DATA_BLOCK "LT"   // DB201
{ S7_Optimized_Access := 'FALSE' }
VERSION : 0.0
// --------------------------------------------------------------------------------
//     program     :    LT
//     description :    define all LT values       
//     name        :    G. Eibelsh鋟ser
//     date        :    26.10.2007
// 
//     revision    :   
//     name        :   
//     date        :    
// 
//                     (c)PVA TePla AG       
//     --------------------------------------------------------------------------------
   VAR
      MOD_AUTO : Bool;   // word 0
      MOD_MANUAL : Bool;
      MOD_SERVICE : Bool;
      MOD_SEMI_AUTO : Bool;
      MOD_START : Bool;
      MOD_CONTINUE : Bool;
      MOD_STOP : Bool;
      SPARE_0_7 : Bool;
      MOD_PUMP_DOWN : Bool;
      MOD_MELTING : Bool;
      MOD_DIP : Bool;
      MOD_NECK : Bool;
      MOD_SHOULDER : Bool;
      MOD_BODY : Bool;
      MOD_ENDCONE : Bool;
      MOD_REMOVAL : Bool;
      MOD_SHUT_DOWN : Bool;   // word 1
      MOD_EMG : Bool;
      SPARE_2_2 : Bool;
      SPARE_2_3 : Bool;
      SPARE_2_4 : Bool;
      SPARE_2_5 : Bool;
      SPARE_2_6 : Bool;
      SPARE_2_7 : Bool;
      SMI_XT_SPD_ON : Bool;
      SMI_XT_ROT_ON : Bool;
      SMI_CR_SPD_ON : Bool;
      SMI_CR_ROT_ON : Bool;
      SMI_HTR_1_ON : Bool;
      SMI_HTR_2_ON : Bool;
      SMI_GAS_FLW_ON : Bool;
      SMI_GAS_PRS_ON : Bool;
      SMI_SI_FDR_ON : Bool;   // word 2
      SMI_DOP_FDR_ON : Bool;
      SMI_MAG_ON : Bool;
      SMI_CR_SPD_COF_ON : Bool;
      SMI_MOB_FDR_ON : Bool;
      SPARE_4_5 : Bool;
      SPARE_4_6 : Bool;
      SPARE_4_7 : Bool;
      XT_LFT_UP : Bool;
      XT_LFT_DN : Bool;
      XT_LFT_FST : Bool;
      XT_ROT_CW : Bool;
      XT_ROT_CCW : Bool;
      XT_ROT_OFF : Bool;
      XT_LFT_OFF : Bool;
      CCZ_OP_ON : Bool;
      CR_LFT_UP : Bool;   // word 3
      CR_LFT_DN : Bool;
      CR_LFT_FST : Bool;
      CR_ROT_CW : Bool;
      CR_ROT_CCW : Bool;
      CR_ROT_OFF : Bool;
      CR_LFT_OFF : Bool;
      SPARE_6_7 : Bool;
      HTR_1_ON : Bool;
      HTR_2_ON : Bool;
      MAG_ON : Bool;
      P2_ON : Bool;
      SI_CRG_WGT_VALID : Bool;
      MAG_STBY_ON : Bool;
      DBL_ALM_SND : Bool;
      CTL_AV_CRUC_ROT_ON : Bool;
      CTL_DIA_ON : Bool;   // word 4
      CTL_GRO_ON : Bool;
      CTL_LVL_ON : Bool;
      CTL_AV_SPD_ON : Bool;
      CTL_HTR_1_TMP_ON : Bool;
      CTL_MELT_TMP_1_ON : Bool;
      CTL_HTR_2_TMP_ON : Bool;
      CTL_MELT_TMP_2_ON : Bool;
      CTL_PRS_ON : Bool;
      V1_OPEN_REQ : Bool;
      V1_CLOSE_REQ : Bool;
      V7_OPEN : Bool;
      V7_CLOSE : Bool;
      V2_1_SEL : Bool;
      V2_2_SEL : Bool;
      V2_X_SEL : Bool;
      V1_OPEN : Bool;   // word 5
      V2_1_OPEN : Bool;
      V3_OPEN : Bool;
      V4_OPEN : Bool;
      V5_OPEN : Bool;
      V6_OPEN : Bool;
      V8_OPEN : Bool;
      V11_OP : Bool;
      V12_OPEN : Bool;
      V2_2_OPEN : Bool;
      V9_1_OPEN : Bool;
      V9_2_OPEN : Bool;
      V1_LS_OPEN : Bool;
      V1_LS_CLOSE : Bool;
      P1_ON : Bool;
      P3_ON : Bool;
      MCC_ON : Bool;   // word 6
      MCC_TST_ON : Bool;
      LSR_ON : Bool;
      LSR_OFF : Bool;
      V16_1_OPEN : Bool;
      V16_2_OPEN : Bool;
      V21_OPEN : Bool;
      CAM_RST_THR_ADJ_ENB : Bool;
      CAM_OFF : Bool;
      CAM_MLT : Bool;
      CAM_DIP : Bool;
      CAM_DIA : Bool;
      CAM_INIT : Bool;
      CAM_SEL_1 : Bool;
      CAM_SEL_2 : Bool;
      CAM_RST_THR_ADJ_DIS : Bool;
      PNBDY : Bool;   // word 7
      BYRST : Bool;
      SUTDN : Bool;
      LEN2_CALC : Bool;
      PMELT : Bool;
      XT_MELT_CONTACT : Bool;
      ALARM : Bool;
      VAC_FNC : Bool;
      VAC_GAT : Bool;
      CLF_APS : Bool;
      CGT_APS : Bool;
      OP_CALL_ON : Bool;
      OP_CALL_ALM : Bool;
      LSR_FIL_LOW : Bool;
      LSR_FIL_HI : Bool;
      LSR_LVL_ABV_REF : Bool;
      FDR_HOP_CON : Bool;   // word 8
      FDR_APS : Bool;
      FDR_LS_TUBE_IN : Bool;
      FDR_LS_TUBE_OUT : Bool;
      FDR_TUBE_DRV_IN : Bool;
      FDR_TUBE_DRV_OUT : Bool;
      FDR_TUBE_DRV_OFF : Bool;
      FDR_FLP_CTL_ON : Bool;
      FDR_FLP_CTL_OFF : Bool;
      XT_DRP_OUT_PRT_OP : Bool;
      XT_DRP_OUT_PRT_CL : Bool;
      XT_DRP_OUT_PRT_ENB : Bool;
      V11_CL : Bool;
      V3_2_OP : Bool;
      V24_OP : Bool;
      PRC_RUN_DONE : Bool;
      CAM_ISP_ON : Bool;   // word 9
      EMG_MOD_REQ : Bool;
      MA_NOT_AVL : Bool;
      NOT_ACKN_ALM : Bool;
      V13_OPEN : Bool;
      V14_OPEN : Bool;
      V15_OPEN : Bool;
      V17_OPEN : Bool;
      V18_OPEN : Bool;
      V19_OPEN : Bool;
      V20_OPEN : Bool;
      V22_OPEN : Bool;
      V23_OPEN : Bool;
      VAC_LINE_IS_OPEN : Bool;
      AUX_FIL_ENB : Bool;
      CAM_PRD_1_SEL : Bool;
      CAM_PRD_2_SEL : Bool;   // word 10
      V25_OPEN : Bool;
      SI_FIL_FSH_SEQ_ON : Bool;
      EDIT_INGOT_ID : Bool;
      EDIT_CARRIER_ID : Bool;
      ENB_LOADING : Bool;
      SMI_GAP_ON : Bool;
      LSR_SEN_PWR_ON : Bool;
      RST_SIHI_PU : Bool;
      RST_HTR_1_PWR_SPL : Bool;
      RST_HTR_2_PWR_SPL : Bool;
      AUTO_OP_CALL : Bool;
      EXT_ACQ_TRG_ON : Bool;
      CAM_CAL : Bool;
      SPARE_21_6 : Bool;
      SPARE_21_7 : Bool;
      CTL_MLT_DRIFT_ON : Bool;   // word 11
      RST_MLT_LVL : Bool;
      MSR_MLT_VIB_ON : Bool;
      SPARE_22_3 : Bool;
      SPARE_22_4 : Bool;
      SPARE_22_5 : Bool;
      SPARE_22_6 : Bool;
      SPARE_22_7 : Bool;
      TEST_CTRL_ON : Bool;
      TEST_CTRL_RST : Bool;
      EMG_ON : Bool;
      SPARE_23_3 : Bool;
      SPARE_23_4 : Bool;
      SPARE_23_5 : Bool;
      BY_FIL_APS : Bool;
      FIL_APS : Bool;
      V3_0_OPEN : Bool;   // word 12
      V3_1_OPEN : Bool;
      XT_LFT_REF_RUN : Bool;
      CR_LFT_REF_RUN : Bool;
      XT_LFT_REF_DONE : Bool;
      CR_LFT_REF_DONE : Bool;
      XT_LFT_REL_LS : Bool;
      CR_LFT_REL_LS : Bool;
      MOB_FDR_IN_POS : Bool;
      MOB_FDR_DCK_ATV : Bool;
      MOB_FDR_UDCK_ATV : Bool;
      MOB_FDR_DCK_DONE : Bool;
      MOB_FDR_UDCK_DONE : Bool;
      MOB_FDR_CH_FDG_POS : Bool;
      ACC_OVP_TEST_ENB : Bool;
      ACC_OVP_OK : Bool;
      MOB_FDR_MVE_IN_SEQ_ON : Bool;   // word 13
      MOB_FDR_MVE_OUT_SEQ_ON : Bool;
      MOB_FDR_MVE_SEQ_ARB : Bool;
      MOB_FDR_VIB_ON : Bool;
      MOB_FDR_CH_HOME_POS : Bool;
      MOB_FDR_TUBE_HOME_POS : Bool;
      MOB_FDR_TUBE_FCH_POS : Bool;
      MOB_FDR_TUBE_FDG_POS : Bool;
      MOB_FDR_EL_CON_DONE : Bool;
      ACC_OVP_TEST_ON : Bool;
      ACC_SC_WTR_STR_ON : Bool;
      ACC_SC_WTR_STR_ENB : Bool;
      SHOW_HTR_1_TRG_TMP : Bool;
      SHOW_XT_RMV_BTN : Bool;
      ENB_KEY_NEXT_MLT_STEP : Bool;
      CTL_FDG_RTE_ON : Bool;
      MOB_FDR_SRV_ON : Bool;
      MOB_FDR_TUBE_UP : Bool;
      MOB_FDR_TUBE_DN : Bool;
      MOB_FDR_TUBE_STOP : Bool;
      MOB_FDR_CH_SW_R : Bool;
      MOB_FDR_CH_SW_L : Bool;
      MOB_FDR_CH_SW_STOP : Bool;
      SH_MLT_LVL_SFT_RUN : Bool;
      ARR_ID_PD : Bool;
      ARR_PD_ID : Bool;
      ARR_PD_ME : Bool;
      ARR_EC_SD : Bool;
      ARR_BY_RE : Bool;
      ARR_EC_RE : Bool;
      ARR_RE_DI : Bool;
      TCH_HOOK_1_ABV : Bool;
      TCH_HOOK_2_ABV : Bool;   // word 15
      TCH_HOOK_3_ABV : Bool;
      TCH_HOOK_4_ABV : Bool;
      TCH_HOOK_1_BLW : Bool;
      TCH_HOOK_2_BLW : Bool;
      TCH_HOOK_3_BLW : Bool;
      TCH_HOOK_4_BLW : Bool;
      GCH_SWD_IN : Bool;
      GCH_SWD_OUT : Bool;
      TCH_CON_GCH : Bool;
      CUF_CLP_LS_SWV_IN_1 : Bool;
      CUF_CLP_LS_SWV_OUT_1 : Bool;
      CUF_CLP_LS_SWV_IN_2 : Bool;
      CUF_CLP_LS_SWV_OUT_2 : Bool;
      HND_LFT_UP : Bool;
      HND_LFT_DN : Bool;
      GCH_SWV_IN : Bool;   // word 16
      GCH_SWV_OUT : Bool;
      MAG_RAI_ON : Bool;
      MAG_LOW_ON : Bool;
      CTL_GAP_ON : Bool;
      SPARE_32_5 : Bool;
      SPARE_32_6 : Bool;
      SPARE_32_7 : Bool;
      SPARE_33_0 : Bool;
      SPARE_33_1 : Bool;
      SPARE_33_2 : Bool;
      SPARE_33_3 : Bool;
      SPARE_33_4 : Bool;
      SPARE_33_5 : Bool;
      SPARE_33_6 : Bool;
      SPARE_33_7 : Bool;
      SPARE : Array[34..63] of Byte;
      XT_HDL_SEQ_MOD : Bool;
      XT_HDL_SEQ_XT_OUT : Bool;
      XT_HDL_SEQ_LD_CRU : Bool;
      XT_HDL_SEQ_HDL_HZ : Bool;
      XT_HDL_OP_CONT : Bool;
      ABORT_FIL_CLN : Bool;
      MLT_GAP_SEARCH : Bool;
      V7_CLN : Bool;
      V7_SW_OUT : Bool;
      V7_SW_IN : Bool;
      V7_LFT_UP : Bool;
      V7_LFT_DN : Bool;
      V7_LFT_UP_REL : Bool;
      V7_LFT_DN_REL : Bool;
      V7_SW_OUT_REL : Bool;
      V7_SW_IN_REL : Bool;
      BEL_LFT_UP_REL : Bool;   // Freigabe
      BEL_LFT_DN_REL : Bool;
      GCH_LFT_UP_REL : Bool;
      GCH_LFT_DN_REL : Bool;
      GCH_SW_OUT_REL : Bool;
      GCH_SW_IN_REL : Bool;
      GCH_SW_LOCKED : Bool;
      TCH_LFT_UP_REL : Bool;
      TCH_LFT_DN_REL : Bool;
      TCH_SW_OUT_REL : Bool;
      TCH_SW_IN_REL : Bool;
      TCH_SW_LOCKED : Bool;
      TCH_TILT_0_REL : Bool;
      TCH_TILT_30_REL : Bool;
      TEC_FLG_LFT_UP_REL : Bool;
      TEC_FLG_LFT_DN_REL : Bool;
      TEC_FLG_SW_OUT_REL : Bool;
      TEC_FLG_SW_IN_REL : Bool;
      TEC_FLG_SW_UNLOCK : Bool;
      UP_FCH_SW_OUT_REL : Bool;
      UP_FCH_SW_IN_REL : Bool;
      UP_FCH_SW_UNLOCK : Bool;
      LO_FCH_SW_OUT_REL : Bool;
      LO_FCH_SW_IN_REL : Bool;
      LO_FCH_SW_UNLOCK : Bool;
      FCH_LFT_UP_REL : Bool;
      FCH_LFT_DN_REL : Bool;
      FCH_HOOK_WORK_REL : Bool;
      FCH_HOOK_HOME_REL : Bool;
      MAG_LFT_UP_REL : Bool;
      MAG_LFT_DN_REL : Bool;
      RESET_ERR_HTR_ETH : Bool;
      SPARE_70_0 : Bool;
      SPARE_70_1 : Bool;
      SPARE_70_2 : Bool;
      SPARE_70_3 : Bool;
      SPARE_70_4 : Bool;
      SPARE_70_5 : Bool;
      SPARE_70_6 : Bool;
      SPARE_70_7 : Bool;
      BEL_LFT_UP : Bool;   // light signals for drives
      BEL_LFT_DN : Bool;
      GCH_LFT_UP : Bool;
      GCH_LFT_DN : Bool;
      TCH_LFT_UP : Bool;
      TCH_LFT_DN : Bool;
      TCH_TILT_0 : Bool;
      TCH_TILT_30 : Bool;
      TEC_FLG_LFT_UP : Bool;
      TEC_FLG_LFT_DN : Bool;
      FCH_LFT_UP : Bool;
      FCH_LFT_DN : Bool;
      MAG_LFT_UP : Bool;
      MAG_LFT_DN : Bool;
      SPARE_72_6 : Bool;
      SPARE_72_7 : Bool;
      GCH_BEL_UP : Bool;   // signals for position of parts
      GCH_BEL_DN : Bool;
      GCH_UP : Bool;
      GCH_DN : Bool;
      GCH_IN : Bool;
      GCH_CLN : Bool;
      GCH_OUT : Bool;
      TCH_UP : Bool;
      TCH_DN : Bool;
      TCH_IN : Bool;
      TCH_CLN : Bool;
      TCH_OUT : Bool;
      TCH_TILT_POS_0 : Bool;
      TCH_TILT_POS_30 : Bool;
      TEC_FLG_SW_OUT : Bool;
      TEC_FLG_SW_IN : Bool;
      UP_FCH_SW_OUT : Bool;
      UP_FCH_SW_IN : Bool;
      LO_FCH_SW_OUT : Bool;
      LO_FCH_SW_IN : Bool;
      GCH_SW_UNLOCK : Bool;
      TCH_SW_UNLOCK : Bool;
      FCH_HOOK_WORK : Bool;
      FCH_HOOK_HOME : Bool;
      MAG_UP : Bool;
      MAG_DN : Bool;
      SPARE_76_2 : Bool;
      SPARE_76_3 : Bool;
      XT_HDL_LFT_DN_REL : Bool;
      XT_HDL_LFT_UP_REL : Bool;
      XT_HDL_SW_OUT_REL : Bool;
      XT_HDL_SW_IN_REL : Bool;
      XT_SLID_FW_REL : Bool;
      XT_SLID_BW_REL : Bool;
      XT_TILT_90_REL : Bool;
      XT_TILT_75_REL : Bool;
      SPARE_77_4 : Bool;
      SPARE_77_5 : Bool;
      SPARE_77_6 : Bool;
      SPARE_77_7 : Bool;
      XT_HDL_LFT_DN : Bool;
      XT_HDL_LFT_UP : Bool;
      XT_HDL_SW_OUT : Bool;
      XT_HDL_SW_IN : Bool;
      XT_SLID_BW : Bool;
      XT_SLID_MID : Bool;
      XT_SLID_FW : Bool;
      XT_TILT_90 : Bool;
      XT_TILT_75 : Bool;
      UP_XT_CLP_CL : Bool;
      UP_XT_CLP_OP : Bool;
      LO_XT_CLP_CL : Bool;
      LO_XT_CLP_OP : Bool;
      SPARE_79_5 : Bool;
      LS_XT_HDL_SW_OUT : Bool;
      LS_XT_HDL_SW_IN : Bool;
      LS_XT_SLID_BW : Bool;
      LS_XT_SLID_MID : Bool;
      LS_XT_SLID_FW : Bool;
      LS_XT_TILT_90 : Bool;
      LS_XT_TILT_75 : Bool;
      LS_UP_XT_CLP_CL : Bool;
      LS_UP_XT_CLP_OP : Bool;
      LS_LO_XT_CLP_CL : Bool;
      LS_LO_XT_CLP_OP : Bool;
      LS_XT_DRP_OUT_PRT_CL : Bool;
      LS_XT_DRP_OUT_PRT_OP : Bool;
      XT_DRP_OUT_PRT_REL : Bool;
      UP_XT_CLP_CL_REL : Bool;
      UP_XT_CLP_OP_REL : Bool;
      LO_XT_CLP_CL_REL : Bool;
      LO_XT_CLP_OP_REL : Bool;
      XT_HDL_LFT_REF_RUN : Bool;
      XT_HDL_LFT_REF_DONE : Bool;
      XT_HDL_SW_REF_RUN : Bool;
      XT_HDL_SW_REF_DONE : Bool;
      XT_HDL_SW_LOCKED : Bool;
      XT_HDL_SW_UNLOCKED : Bool;
      LS_UP_XT_CLP_PLATE : Bool;
      XT_HDL_CLP_OP_CONT : Bool;
      XT_HDL_CUT_OP_CONT : Bool;
      HOI_TOOL_INST : Bool;
      HOI_TOOL_CRU_INS : Bool;
      LD_CRU_OP_CONT : Bool;
      LD_CRU_FIN : Bool;
      HOI_TOOL_UNIS : Bool;
      HOI_TOOL_HZ_INS : Bool;
      LD_HZ_OP_CONT : Bool;
      LD_HZ_FIN : Bool;
      SI_FIL_RDY : Bool;
      MP_SERVICE : Bool;
      V2_11_OPEN : Bool;
      V1_1_OPEN : Bool;
      V3_3_OPEN : Bool;
      V3_4_OPEN : Bool;
      V22_1_OPEN : Bool;
      SPARE_OP : Array[82..127] of Byte;
   END_VAR
BEGIN
END_DATA_BLOCK

DATA_BLOCK "DIS"   // DB202
{ S7_Optimized_Access := 'FALSE' }
VERSION : 0.0
// --------------------------------------------------------------------------------
//     program     :    DIS
//     description :    define all DIS values       
//     name        :    G. Eibelsh鋟ser
//     date        :    26.10.2007
// 
//     revision    :
//     name        :
//     date        :    
//                     (c)PVA TePla AG       
//     --------------------------------------------------------------------------------
   VAR
      SET_XT_SPD : Real;   // dword 0
      ACT_XT_SPD : Real;
      SET_XT_ROT : Real;
      ACT_XT_ROT : Real;
      ACT_XT_POS : Real;
      SET_CR_SPD : Real;
      ACT_CR_SPD : Real;
      SET_CR_ROT : Real;
      ACT_CR_ROT : Real;   // dword 32
      ACT_CR_POS : Real;
      SET_HTR_1_PWR : Real;
      ACT_HTR_1_PWR : Real;
      SET_HTR_1_TMP : Real;
      ACT_HTR_1_TMP : Real;
      ACT_HTR_1_AV_TMP : Real;
      ACT_HTR_1_CUR : Real;
      ACT_HTR_1_VLT : Real;   // dword 64
      ACT_HTR_1_RES : Real;
      SET_HTR_1_TMP_INC : Real;
      ACT_HTR_1_TMP_INC : Real;
      SET_HTR_2_PWR : Real;
      ACT_HTR_2_PWR : Real;
      SET_HTR_2_TMP : Real;
      ACT_HTR_2_TMP : Real;
      ACT_HTR_2_AV_TMP : Real;   // dword 96
      ACT_HTR_2_CUR : Real;
      ACT_HTR_2_VLT : Real;
      ACT_HTR_2_RES : Real;
      SET_HTR_2_PWR_INC : Real;
      ACT_HTR_2_PWR_INC : Real;
      SET_MAG_1_CUR : Real;
      ACT_MAG_1_CUR : Real;
      ACT_MAG_1_VLT : Real;   // dword 128
      ACT_MAG_1_RES : Real;
      SET_MAG_2_CUR : Real;
      ACT_MAG_2_CUR : Real;
      ACT_MAG_2_VLT : Real;
      ACT_MAG_2_RES : Real;
      SET_GAS_1_FLW : Real;
      ACT_GAS_1_FLW : Real;
      SET_GAS_2_FLW : Real;   // dword 160
      ACT_GAS_2_FLW : Real;
      SET_PRS_FNC : Real;
      HTR_1_TMP_SET_PHA_STR : Real;   // heater 1 temperature setpoint at phase start
      HTR_2_PWR_SET_PHA_STR : Real;   // heater 2 power setpoint at phase start
      ACT_TOT_XT_LGH : Real;   // actual total crystal lenght (neck, shoulder, body, endcone)
      ACT_PRS_DROP_FDR : Real;
      ACT_PRS_CLF : Real;   // actual pressure furnace
      ACT_PRS_CGT : Real;   // dword 192 // actual pressure gate
      ACT_PRS_FDR : Real;   // actual pressure feeder
      SET_CTL_VALVE_POS : Real;
      ACT_LEAKR_FNC : Real;
      ACT_LEAKR_FDR : Real;
      SET_XT_DIA : Real;
      ACT_XT_DIA : Real;
      SET_XT_AV_SPD : Real;
      ACT_XT_AV_SPD : Real;   // dword 224
      SET_LSR_MLT_LVL : Real;
      ACT_LSR_MLT_LVL : Real;
      SET_XTAL_GRO : Real;
      ACT_XTAL_GRO : Real;
      SET_MLT_TMP_1 : Real;
      ACT_MLT_TMP_1 : Real;
      SET_AVG_CRUC_ROT : Real;
      ACT_AVG_CRUC_ROT : Real;   // dword 256
      ACT_XT_GROSS_WGT : Real;
      ACT_PER_BGT_AREA : Real;
      ACT_AMT_BLOBS : Real;
      CALC_THR : Real;
      ACT_XT_LEN_MM : Real;
      ACT_XT_LEN_PERC : Real;
      ACT_XT_WGT_MEAS : Real;
      ACT_XT_WGT_CALC : Real;   // dword 288
      ACT_PLC_VERSION : Real;
      ACT_PLC_CONFIG : Real;
      ACT_BDY2_LEN : Real;
      ACT_CR_POS_DIPPING : Real;
      ACT_CGT_LFT_POS : Real;
      ACT_CGT_SWL_POS : Real;
      ACT_SI_CRG_WGT : Real;
      ACT_CA_DIA_PIX : Real;   // dword 320
      ACT_XT_LEN_BY2_RP : Real;
      SET_HTR_1_PWR_INC : Real;
      ACT_HTR_1_PWR_INC : Real;
      ACT_TME_TILL_EMG : Real;
      ACT_PLT_HDW_ID : Real;
      ACT_PHA_STA : Real;
      ACT_SMI_STA : Real;
      ACT_WTR_TMP_PWR_CAB : Real;   // dword 352
      ACT_WTR_FLW_PWR_CAB : Real;
      ACT_WTR_TMP_CUR_FEED : Real;
      ACT_WTR_FLW_CUR_FEED : Real;
      ACT_WTR_TMP_PLT : Real;
      ACT_WTR_FLW_PLT : Real;
      ACT_WTR_TMP_GCH : Real;
      ACT_WTR_FLW_GCH : Real;
      ACT_WTR_TMP_GCH_V : Real;   // dword 384
      ACT_WTR_FLW_GCH_V : Real;
      ACT_WTR_TMP_CR_SFT : Real;
      ACT_WTR_FLW_CR_SFT : Real;
      ACT_WTR_TMP_HTR_1 : Real;
      ACT_WTR_FLW_HTR_1 : Real;
      ACT_WTR_TMP_CFT_2 : Real;
      ACT_WTR_FLW_CFT_2 : Real;
      ACT_WTR_TMP_GATE : Real;   // dword 416
      ACT_WTR_FLW_GATE : Real;
      ACT_WTR_TMP_SPC : Real;
      ACT_WTR_FLW_SPC : Real;
      ACT_WTR_TMP_VSL : Real;
      ACT_WTR_FLW_VSL : Real;
      ACT_WTR_TMP_FCH : Real;
      ACT_WTR_FLW_FCH : Real;
      ACT_WTR_TMP_TCH : Real;   // dword 448
      ACT_WTR_FLW_TCH : Real;
      ACT_XT_WGT_RTE : Real;
      ACT_XT_DIA_CALC : Real;
      ACT_CTL_VALVE_POS : Real;
      ACT_GEAR_OIL_TMP_P1 : Real;
      ACT_COOLANT_TMP_P1 : Real;
      ACT_VIB_P1 : Real;
      ACT_WTR_TMP_VPTS : Real;   // dword 480
      ACT_WTR_FLW_VPTS : Real;
      ACT_INPUT_SIMOCODE_P1 : Real;
      ACT_INPUT_SIMOCODE_P2 : Real;
      ACT_FNC_PRS_BEF_LKT : Real;
      ACT_CAM_THR : Real;
      ACT_XT_ORB : Real;
      ACT_MLT_LVL : Real;
      TEST_P_PART_OUT : Real;   // dword 512
      TEST_I_PART_OUT : Real;
      TEST_D_PART_OUT : Real;
      TEST_CTRL_OUT : Real;
      ACT_PRD_2_CTR_X : Real;
      ACT_PRD_2_CTR_Y : Real;
      AVG_PRD_2_CTR_X : Real;
      AVG_PRD_2_CTR_Y : Real;
      XT_LFT_ERR_CODE : Real;   // dword 544
      XT_ROT_ERR_CODE : Real;
      CR_LFT_ERR_CODE : Real;
      CR_ROT_ERR_CODE : Real;
      ACT_MLT_VIB : Real;
      ACT_MLT_VIB_RAW : Real;
      MOB_FDR_ACT_TUBE_TMP : Real;
      MOB_FDR_SET_VIB_FRQ : Real;
      SET_CR_SPD_COF_OFFS : Real;   // dword 576
      SET_CR_SPD_COF : Real;
      EFF_XT_SPD_BY : Real;
      TOT_MAN_OP_TIME : Real;
      ACT_WTR_TMP_PU : Real;
      ACT_WTR_FLW_PU : Real;
      ACT_MAG_STATE : Real;
      MOB_FDR_ACT_TUBE_POS : Real;
      ACC_WTR_TMP : Real;   // dword 608
      ACC_WTR_PRS_IN : Real;
      ACC_WTR_FLW_OUT : Real;
      ACC_WTR_FLW_IN : Real;
      DIST_MELT_FUN : Real;
      ACT_WTR_FLW_RING : Real;
      ACT_WTR_TMP_RING : Real;
      MOB_FDR_ACT_CRG_LVL : Real;
      TOT_GAS_CSP : Real;   // dword 640
      TOT_PWR_CSP : Real;
      ACC_TC : Real;
      ACC_WTR_DIFF : Real;
      ACT_DIA_PTS_INCL : Real;
      ACT_MAG_FLD : Real;
      ACT_MAG_1_TMP : Real;
      ACT_MAG_2_TMP : Real;
      HND_LFT_ERR_CODE : Real;   // dword 672
      P1 : Real;
      P3 : Real;
      V2_1 : Real;
      V21 : Real;
      V22 : Real;
      V3 : Real;
      V4 : Real;
      V5 : Real;   // dword 704
      V6 : Real;
      PRS_CTRL : Real;
      XT_LFT : Real;
      XT_ROT : Real;
      CR_LFT : Real;
      CR_ROT : Real;
      HTR_1 : Real;
      TMP_CTRL : Real;   // dword 736
      CAM_CTRL : Real;
      CAM_MELT : Real;
      CAM_DIP : Real;
      CAM_DIA : Real;
      MCC : Real;
      MCC_TEST : Real;
      FILTER_CLEAN : Real;
      MLT_LVL_CTRL : Real;   // dword 768
      GATE_V : Real;
      GCH_OP : Real;
      TCH_OP : Real;
      FCH_OP : Real;
      ME_TMP_OFFS : Real;
      ACC_WTR_SPL_PRS : Real;
      V24 : Real;
      V3_2 : Real;   // dword 800
      ME_UP_CR_POS_LIM : Real;
      RE_HTR_1_TRG_SET_TMP : Real;
      ACT_MAG_POS : Real;
      ACT_HND_LFT_MOT_ROT : Real;
      ACT_HND_LFT_MOT_CUR : Real;
      ACT_STB_NE_LEN : Real;
      CALC_SH_TRS_DIA : Real;
      ACT_STB_NE_LEN_PRC : Real;   // dword 832
      PWR_CTR_PWR : Real;
      PWR_CTR_COSPHI : Real;
      PWR_CTR_CONSUM : Real;
      PWR_CTR_VLT_L1_2 : Real;
      PWR_CTR_VLT_L2_3 : Real;
      PWR_CTR_VLT_L3_1 : Real;
      PWR_CTR_CUR_L1 : Real;
      PWR_CTR_CUR_L2 : Real;   // dword 864
      PWR_CTR_CUR_L3 : Real;
      MOB_FDR_ACT_VIB_FRQ : Real;
      MOB_FDR_OFFS_VIB_FRQ : Real;
      MOB_FDR_CUTE_WGT : Real;
      MOB_FDR_CUTE_WGT_TAR : Real;
      ACT_STD_DEV_FILL_LVL : Real;
      ACT_FDG_RTE : Real;
      SET_FDG_RTE : Real;   // dword 896
      ACT_MLT_GAP_OFFS : Real;
      ACT_XT_WGT_RTE_MM : Real;
      ACT_CUR_P1 : Real;
      S_CAM_ACT_XT_DIA : Real;
      S_CAM_ACT_MLT_LVL_CHG : Real;
      SET_SPEED_OFFS : Real;   // actual controller output
      SET_GAP_CTL_OFFS : Real;   // actual controller output
      FI_DIA_NE_T1 : Real;   // dword 928
      FI_DIA_SH_T1 : Real;
      FI_DIA_BY_T1 : Real;
      FI_DIA_NE_T2 : Real;
      FI_DIA_SH_T2 : Real;
      FI_DIA_BY_T2 : Real;
      FI_GRO_SH : Real;
      ACT_XT_WGT_DLY_T1 : Real;
      FI_TMP_HTR_1 : Real;   // dword 960
      FI_AV_TMP_1 : Real;
      FI_MLT_TMP_1 : Real;
      FI_AV_SPD : Real;
      FI_SH_AV_CRUC_ROT : Real;
      FI_BY_AV_CRUC_ROT : Real;
      CTL_AVG_SPD_OFFS_TF : Real;
      ACT_WGT_LC_BRUTTO : Real;
      CTL_HTR_1_TMP_GN : Real;   // dword 992
      CTL_HTR_1_TMP_TI : Real;
      CTL_HTR_1_TMP_TD : Real;
      CTL_HTR_1_TMP_T1 : Real;
      CTL_HTR_1_TMP_GN_DIP : Real;
      CTL_HTR_1_TMP_TI_DIP : Real;
      CTL_HTR_1_TMP_TD_DIP : Real;
      CTL_HTR_1_TMP_T1_DIP : Real;
      CTL_PRS_GN : Real;   // dword 1024
      CTL_PRS_TI : Real;
      CTL_PRS_TD : Real;
      CTL_PRS_T1 : Real;
      CTL_PRS_GN_HI : Real;
      CTL_PRS_TI_HI : Real;
      CTL_PRS_TD_HI : Real;
      CTL_PRS_T1_HI : Real;
      CTL_MLT_DRIFT_GN : Real;   // dword 1056
      CTL_MLT_DRIFT_TI : Real;
      CTL_MLT_DRIFT_TD : Real;
      CTL_MLT_DRIFT_T1 : Real;
      CTL_MLT_TMP_GN : Real;
      CTL_MLT_TMP_TI : Real;
      CTL_MLT_TMP_TD : Real;
      CTL_MLT_TMP_T1 : Real;
      CTL_DIA_GN : Real;   // dword 1088
      CTL_DIA_TI : Real;
      CTL_DIA_TD : Real;
      CTL_DIA_T1 : Real;
      CTL_AV_SPD_GN : Real;
      CTL_AV_SPD_TI : Real;
      CTL_AV_SPD_TD : Real;
      CTL_AV_SPD_T1 : Real;
      CTL_GRO_GN : Real;   // dword 1120
      CTL_GRO_TI : Real;
      CTL_GRO_TD : Real;
      CTL_GRO_T1 : Real;
      CTL_AV_CRUC_ROT_GN : Real;
      CTL_AV_CRUC_ROT_TI : Real;
      CTL_AV_CRUC_ROT_TD : Real;
      CTL_AV_CRUC_ROT_T1 : Real;
      CTL_DIA_TMP_GN : Real;   // dword 1152
      CTL_DIA_TMP_TI : Real;
      CTL_DIA_TMP_TD : Real;
      CTL_DIA_TMP_T1 : Real;
      CTL_AV_OFFS_GN : Real;
      CTL_AV_OFFS_TI : Real;
      CTL_AV_OFFS_TD : Real;
      CTL_AV_OFFS_T1 : Real;
      CTL_OFFS_SPEED_GN : Real;   // dword 1184
      CTL_OFFS_SPEED_TI : Real;
      CTL_OFFS_SPEED_TD : Real;
      CTL_OFFS_SPEED_T1 : Real;
      CTL_GAP_GN : Real;
      CTL_GAP_TI : Real;
      CTL_GAP_TD : Real;
      CTL_GAP_T1 : Real;
      ACT_WTR_TMP_TEC_FLG : Real;   // dword 1216
      ACT_WTR_FLW_TEC_FLG : Real;
      ACT_WTR_TMP_UP_FCH : Real;
      ACT_WTR_FLW_UP_FCH : Real;
      ACT_WTR_TMP_XT_SFT : Real;
      ACT_WTR_FLW_XT_SFT : Real;
      ACT_WTR_TMP_GCH_H : Real;
      ACT_WTR_FLW_GCH_H : Real;   // dword 1248
      ACT_WTR_TMP_SOC_BCH : Real;
      ACT_WTR_FLW_SOC_BCH : Real;
      ACT_WTR_TMP_PWR_CAB2 : Real;
      ACT_WTR_FLW_PWR_CAB2 : Real;
      ACT_WTR_TMP_ACC : Real;
      ACT_WTR_FLW_ACC : Real;
      ACT_WTR_TMP_MAG_CO1 : Real;
      ACT_WTR_FLW_MAG_CO1 : Real;
      ACT_WTR_TMP_MAG_CO2 : Real;   // dword 1280
      ACT_WTR_FLW_MAG_CO2 : Real;
      ACT_WTR_TMP_MAG_CO3 : Real;
      ACT_WTR_FLW_MAG_CO3 : Real;
      ACT_WTR_TMP_MAG_CO4 : Real;
      ACT_WTR_FLW_MAG_CO4 : Real;
      ACT_WTR_TMP_MAG_CAB : Real;
      ACT_WTR_FLW_MAG_CAB : Real;
      ACT_ITL_NO : Real;   // dword 1312
      ACT_ITL_STAT : Real;
      ACT_ITL_CAUSE : Real;
      ACT_TEC_FCH_SW_POS : Real;
      ACT_UP_FCH_SW_POS : Real;
      ACT_LO_FCH_SW_POS : Real;
      ACT_TEC_FLG_LFT_POS : Real;
      ACT_FCH_LFT_POS : Real;
      ACT_POS_XT_HDL_LFT : Real;   // dword 1344
      ACT_POS_XT_HDL_SW : Real;
      XT_HDL_LFT_ERR_CODE : Real;
      XT_HDL_SW_ERR_CODE : Real;
      XT_HDL_CLP_WGT : Real;
      XT_HDL_CLP_WGT_TAR : Real;
      S_CAM_1_ACT_RAD_PT : Real;
      S_CAM_2_ACT_RAD_PT : Real;
      RAW_XT_DIA : Real;   // dword 1376
      RAW_PYR_MELT_TMP : Real;
      RAW_PYR_HTR_1_TMP : Real;
      RAW_SET_XT_SPD : Real;
      DIA_CONT_P : Real;
      DIA_CONT_D : Real;
      DIA_CONT_I : Real;
      HTR_1_CONT_P : Real;
      HTR_1_CONT_D : Real;   // dword 1408
      HTR_1_CONT_I : Real;
      AVG_SPD_CONT_P : Real;
      AVG_SPD_CONT_D : Real;
      AVG_SPD_CONT_I : Real;
      OFFS_SPD_CONT_P : Real;
      OFFS_SPD_CONT_D : Real;
      OFFS_SPD_CONT_I : Real;
      GAP_CONT_P : Real;   // dword 1440
      GAP_CONT_D : Real;
      GAP_CONT_I : Real;
      AVG_GAP_CONT_P : Real;
      AVG_GAP_CONT_D : Real;
      AVG_GAP_CONT_I : Real;
      SET_AVG_GAP_OFFS_T_INC : Real;
      RAW_CAM_DIA_PIX_1 : Real;
      RAW_CAM_DIA_PIX_2 : Real;   // dword 1472
      RAW_CAM_DIA_PIX_3 : Real;
      RAW_CAM_DIA_PIX_4 : Real;
      RAW_CAM_DIA_PIX_5 : Real;
      RAW_CAM_DIA_PIX_6 : Real;
      RAW_CAM_DIA_PIX_7 : Real;
      RAW_CAM_DIA_PIX_8 : Real;
      RAW_CAM_DIA_PIX_9 : Real;
      RAW_CAM_DIA_PIX_10 : Real;   // dword 1504
      ACT_WTR_TMP_GCH_ADDS : Real;
      ACT_WTR_FLW_GCH_ADDS : Real;
      ACT_HTR_1_ETH_FLT_VAL : Real;
      ACT_HTR_2_ETH_FLT_VAL : Real;
      ACT_CTL_VALVE_POS_V1_1 : Real;
      SET_CTL_VALVE_POS_V1_1 : Real;
      ACT_PRS_MAIN_FIL : Real;
      ACT_PRS_BYP_FIL : Real;
      GRW_RTE_CONT_P : Real;
      GRW_RTE_CONT_I : Real;
      GRW_RTE_CONT_D : Real;
      ACT_HTR1_ETH_VLT_PLUS : Real;
      ACT_HTR1_ETH_VLT_MINUS : Real;
      ACT_HTR2_ETH_VLT_PLUS : Real;
      ACT_HTR2_ETH_VLT_MINUS : Real;
      ACT_PRS_AR_VSL : Real;
      PRS_DIFF_FIL_TO_FCH : Real;
      HTR_1_PWR_SET_PHA_STR : Real;
      ACT_TORQ_CR_ROT : Real;
      ACT_WTR_TMP_HLD_ACC : Real;
      ACT_WTR_FLW_HLD_ACC : Real;
      XT_MELT_CONTACT : Real;
      RE_HTR_1_TRG_SET_PWR : Real;
      SET_EFF_XT_SPD : Real;
      ACT_WTR_FLW_VAC_BYP : Real;
      ACT_WTR_TMP_VAC_BYP : Real;
      ACT_WTR_FLW_CONE : Real;
      ACT_WTR_TMP_CONE : Real;
      ACT_SEED_LSR_REF_POS : Real;
      ACT_CR_DIP_POS : Real;
      SPARE_1628 : Real;
      HTR_1_RES_DEV_CNT : Real;
      HTR_2_RES_DEV_CNT : Real;
   END_VAR
BEGIN
END_DATA_BLOCK

DATA_BLOCK "KYA"   // DB203
{ S7_Optimized_Access := 'FALSE' }
VERSION : 0.0
// --------------------------------------------------------------------------------
//     program     :    KYA
//     description :    define all KYA values       
//     name        :    G. Eibelsh鋟ser
//     date        :    26.10.2007
// 
//     revision    :
//     name        :
//     date        :    
//                     (c)PVA TePla AG       
//     --------------------------------------------------------------------------------
   VAR
      SET_XT_SPD : Real;   // dword 0
      SET_XT_ROT : Real;
      SET_CR_SPD : Real;
      SET_CR_ROT : Real;
      SET_HTR_1_PWR : Real;
      SET_HTR_2_PWR : Real;
      SET_HTR_1_TMP : Real;
      SET_HTR_2_TMP : Real;
      SET_MELT_TMP_1 : Real;   // dword 32
      SET_MELT_TMP_2 : Real;
      SET_MAG_1_CUR : Real;
      SET_MAG_2_CUR : Real;
      SET_GAS_1_FLW : Real;
      SET_GAS_2_FLW : Real;
      SET_PRS_FNC : Real;
      SET_CTL_VALVE_POS : Real;
      SET_CAM_THR : Real;   // dword 64
      SET_CAM_WIN_POS_H : Real;
      SET_CAM_WIN_POS_V : Real;
      SET_CAM_WIN_SIZE_H : Real;
      SET_CAM_WIN_SIZE_V : Real;
      SET_DIP_POS_CR : Real;
      ACT_BDY2_LEN : Real;
      SET_OP_CALL_TME : Real;
      SET_XT_LFT_OFS : Real;   // dword 96
      SET_XT_LFT_GN : Real;
      SET_XT_ROT_OFS : Real;
      SET_XT_ROT_GN : Real;
      SET_CR_LFT_OFS : Real;
      SET_CR_LFT_GN : Real;
      SET_CR_ROT_OFS : Real;
      SET_CR_ROT_GN : Real;
      SET_THR_CAL_FACT : Real;   // dword 128
      SET_FDR_FLP_TME_OP : Real;
      SET_FDR_FLP_TME_CL : Real;
      SET_CR_SPD_COF : Real;
      DI_NECK_RMLT_LEN : Real;
      SET_SEN_THR_P1 : Real;
      SET_SEN_THR_P2 : Real;
      SET_SEN_THR_P3 : Real;
      SET_SEN_THR_P4 : Real;   // dword 160
      SET_SEN_CTR_X_P1 : Real;
      SET_SEN_CTR_Y_P1 : Real;
      SET_SEN_WDH_P1 : Real;
      SET_SEN_HGT_P1 : Real;
      SET_SEN_CTR_X_P2 : Real;
      SET_SEN_CTR_Y_P2 : Real;
      SET_SEN_OUT_RAD_P2 : Real;
      SET_SEN_IN_RAD_P2 : Real;   // dword 192
      SET_SEN_SEQ_STR_AGL_P2 : Real;
      SET_SEN_SEQ_STP_AGL_P2 : Real;
      SET_SEN_CTR_X_P3 : Real;
      SET_SEN_CTR_Y_P3 : Real;
      SET_SEN_WDH_P3 : Real;
      SET_SEN_CTR_X_P4 : Real;
      SET_SEN_CTR_Y_P4 : Real;
      SET_SEN_WDH_P4 : Real;   // dword 224
      SET_SEN_HGT_P4 : Real;
      SET_SEN_MLT_VIB_CTR_X : Real;
      SET_SEN_MLT_VIB_CTR_Y : Real;
      SET_SEN_MLT_VIB_WDH : Real;
      SET_MAG_RATIO_CUR : Real;
      SET_SEN_MLT_VIB_THR : Real;
      CALC_WGT_GRW_XT : Real;
      TEST_CTRL_SEL : Real;   // dword 256
      TEST_CTRL_GN : Real;
      TEST_CTRL_I : Real;
      TEST_CTRL_D : Real;
      TEST_CTRL_D_DLY : Real;
      MOB_FDR_SET_VIB_FRQ : Real;
      SET_FDG_RTE : Real;
      SET_GAP_SMI : Real;
      CAM_ACQ_DLY : Real;   // dword 288
      SET_ROI_CTR_X_SCAM : Real;
      SET_ROI_CTR_Y_SCAM : Real;
      SET_ROI_WDH_SCAM : Real;
      SET_ROI_HGT_SCAM : Real;
      SET_CTL_VALVE_POS_V1_1 : Real;
      SET_CAM_2_THR : Real;
      WAIT_TME_WITH_BYP_FIL : Real;
      SPARE_320 : Real;   // dword 320
      SPARE_324 : Real;
      SPARE_328 : Real;
      SPARE_332 : Real;
      SPARE_336 : Real;
      SPARE_340 : Real;
      SPARE_344 : Real;
      SPARE_348 : Real;
      SPARE : Array[352..511] of Byte;
   END_VAR
BEGIN
END_DATA_BLOCK

DATA_BLOCK "STA"   // DB204
{ S7_Optimized_Access := 'FALSE' }
VERSION : 0.0
// --------------------------------------------------------------------------------
//     program     :    STA
//     description :    actual status variables      
//     name        :    G. Eibelsh鋟ser
//     date        :    27.10.2007
// 
//     revision    :
//     name        :
//     date        :    
//                     (c)PVA TePla AG       
//     --------------------------------------------------------------------------------
   VAR
      ACT_PROCESS : Int;   // actual process (ID, PD, ME ...)
      ACT_OP_MSG : Int;   // actual operator message
      ACT_STE_NO : Int;   // active step of apc sequence
      ACT_TME_TOT : DInt;   // total time
      ACT_TME_PROC : DInt;   // process time (for each phase)
      ACT_TME_STE : DInt;   // step time (till end of step)
      DEAD_BAND_PC_ALIVE : Int;   // dead band PC alive
      ACT_STATE : Int;   // actual machine state
      ACT_DATA_LOG_ITV : Int;   // actual datalogging interval
      PRC_STR_TME : Date_And_Time;   // process start time stamp
      PRC_END_TME : Date_And_Time;   // process end time stamp
      ACT_RCP_NAME : String[200];   // actual recipe name
      ACT_INGOT_ID : String[200];   // actual ingot number (ID)
      ACT_DVC_CNF_BYTE_0 : Byte;   // actual hardware device configuration
      ACT_DVC_CNF_BYTE_1 : Byte;   // actual hardware device configuration
      ACT_DVC_CNF_BYTE_2 : Byte;   // actual hardware device configuration
      ACT_DVC_CNF_BYTE_3 : Byte;   // actual hardware device configuration
      ACT_DVT_PRD_NO : Real;   // actual camera product number
      SPARE_REAL_01 : Real;   // spare
      SPARE_REAL_02 : Real;   // spare
      SPARE_REAL_03 : Real;   // spare
      SPARE_REAL_04 : Real;   // spare
      SPARE_REAL_05 : Real;   // spare
      SPARE_REAL_06 : Real;   // spare
      SPARE_REAL_07 : Real;   // spare
      OP_CALL_RMG_MIN : Int;   // operator call remaining minutes
      OP_CALL_RMG_SEC : Int;   // operator call remaining secondsion
      SEMI_E10_STATE : Int;   // machine state according Semi E10
      MAN_SEL_REAS : Int;   // reason of manual selection
      INGOT_ID_TIMEOUT : Int;   // spare
      FEEDER_ID : Int;   // ID No. from mobile Feeder
      SPARE_INT_04 : Int;   // spare
      ACT_CHARGE_ID : String[30];   // actual charge number (ID)
      ACT_CRU_ID : String[30];   // actual cruible number (ID)
      SPARE_STRING_03 : String[30];   // spare
      SPARE_STRING_04 : String[30];   // spare
      USER_NAME : String[30];   // user name
      CARRIER_ID : String[10];   // number of Si transport carrier
      AUX_INFO : String[200];   // auxilliary information from CDP contains ingot ID
      AUX_COMMENT : String[254];   // free editable comment
      AUX_FLAGS : DWord;   // Bit Leiste
      PRC_STR_DATE : Date;   // process start date
      PRC_STR_TIME : Time_Of_Day;   // process start time
      PRC_END_DATE : Date;   // process end date
      PRC_END_TIME : Time_Of_Day;   // process end time
      INTERL_TRIGGER : Bool;   // Interlock Trigger
      INT_STAT : Byte;   // Interlock Byte
      INT_NBR : Int;   // Interlock nummer
      ACT_DVC_CNF_DW : DWord;   // Hardware DW
      ITL_NO : Int;   // spare
      MACHINE_NO : Int;   // Machine number
      BEL_LFT_POS : Int;   // Bellow pos for mobile panel
      GCH_LFT_POS : Int;   // Gate chamber pos for mobile panel
      GCH_SW_POS : Int;   // Gate chamber swivel pos for mobile panel
      TCH_LFT_POS : Int;   // Top chamber pos for mobile panel
      TCH_SW_POS : Int;   // Top chamber swivel pos for mobile panel
      TCH_TILT_POS : Int;   // Top chamber tilt pos for mobile panel
      TEC_FLG_POS : Int;   // Teechn. flange pos for mobile panel
      UP_FCH_LFT_POS : Int;   // Furnace chamber pos for mobile panel
      LO_FCH_LFT_POS : Int;   // Furnace chamber pos for mobile panel
      MAG_LFT_POS : Int;   // Bellow pos for mobile panel
      V7_LFT_POS : Int;
      V7_SW_POS : Int;
      XT_HDL_LFT_POS : Int;
      XT_HDL_SLID_POS : Int;
      SPARE_1180 : Int;
      SPARE_1182 : Int;
      OP_MSG_HDL_SEQ : Int;
      SPARE_INT : Array[0..10] of Int;
   END_VAR
BEGIN
END_DATA_BLOCK

DATA_BLOCK "SM_FLT_NOT_ACKN"   // DB205
{ S7_Optimized_Access := 'FALSE' }
VERSION : 0.0
// --------------------------------------------------------------------------------
//     program     :    SM_FLT_NOT_ACKN
//     description :    List of not acknowledged fault signals      
//     name        :    G. Eibelsh鋟ser
//     date        :    01.12.99
// 
//     revision    :    Anzahl der Alarmworte verdoppelt
//     name        :    G. Eibelsh鋟ser
//     date        :    04.01.2007
//     
//                     (c)PVA TePla AG         
//     --------------------------------------------------------------------------------
   VAR
      ALARM_WORD_0 : Word;   // F001 - F016
      ALARM_WORD_1 : Word;   // F017 - F032
      ALARM_WORD_2 : Word;   // F033 - F048
      ALARM_WORD_3 : Word;   // F049 - F064
      ALARM_WORD_4 : Word;   // F065 - F080
      ALARM_WORD_5 : Word;   // F081 - F096
      ALARM_WORD_6 : Word;   // F097 - F112
      ALARM_WORD_7 : Word;   // F113 - F128
      ALARM_WORD_8 : Word;   // F129 - F144
      ALARM_WORD_9 : Word;   // F145 - F160
      ALARM_WORD_10 : Word;   // F161 - F176
      ALARM_WORD_11 : Word;   // F177 - F192
      ALARM_WORD_12 : Word;   // F193 - F208
      ALARM_WORD_13 : Word;   // F209 - F224
      ALARM_WORD_14 : Word;   // F225 - F240
      ALARM_WORD_15 : Word;   // F241 - F256
      ALARM_WORD_16 : Word;   // F257 - F272
      ALARM_WORD_17 : Word;   // F273 - F288
      ALARM_WORD_18 : Word;   // F289 - F304
      ALARM_WORD_19 : Word;   // F305 - F320
      ALARM_WORD_20 : Word;   // F321 - F336
      ALARM_WORD_21 : Word;   // F337 - F352
      ALARM_WORD_22 : Word;   // F353 - F368
      ALARM_WORD_23 : Word;   // F369 - F384
      ALARM_WORD_24 : Word;   // F385 - F400
      ALARM_WORD_25 : Word;   // F401 - F416
      ALARM_WORD_26 : Word;   // F417 - F432
      ALARM_WORD_27 : Word;   // F433 - F448
      ALARM_WORD_28 : Word;   // F449 - F464
      ALARM_WORD_29 : Word;   // F465 - F480
      ALARM_WORD_30 : Word;   // F481 - F496
      ALARM_WORD_31 : Word;   // F497 - F512
      ALARM_WORD_32 : Word;   // F513 - F528
      ALARM_WORD_33 : Word;   // F529 - F544
      ALARM_WORD_34 : Word;   // F545 - F560
      ALARM_WORD_35 : Word;   // F561 - F576
      ALARM_WORD_36 : Word;   // F577 - F592
      ALARM_WORD_37 : Word;   // F593 - F608
      ALARM_WORD_38 : Word;   // F609 - F624
      ALARM_WORD_39 : Word;   // F625 - F640
      ALARM_WORD_40 : Word;   // F641 - F656
      ALARM_WORD_41 : Word;   // F657 - F672
      ALARM_WORD_42 : Word;   // F673 - F688
      ALARM_WORD_43 : Word;   // F689 - F704
      ALARM_WORD_44 : Word;   // F705 - F720
      ALARM_WORD_45 : Word;   // F721 - F736
      ALARM_WORD_46 : Word;   // F737 - F752
      ALARM_WORD_47 : Word;   // F753 - F768
      ALARM_WORD_48 : Word;   // F769 - F784
      ALARM_WORD_49 : Word;   // F785 - F800
      ALARM_WORD_50 : Word;   // F801 - F816
      ALARM_WORD_51 : Word;   // F817 - F832
      ALARM_WORD_52 : Word;   // F833 - F848
      ALARM_WORD_53 : Word;   // F849 - F864
      ALARM_WORD_54 : Word;   // F865 - F880
      ALARM_WORD_55 : Word;   // F881 - F896
      ALARM_WORD_56 : Word;   // F897 - F912
      ALARM_WORD_57 : Word;   // F913 - F928
      ALARM_WORD_58 : Word;   // F929 - F944
      ALARM_WORD_59 : Word;   // F945 - F960
      ALARM_WORD_60 : Word;   // F961 - F976
      ALARM_WORD_61 : Word;   // F977 - F992
      ALARM_WORD_62 : Word;   // F993 - F1008
      ALARM_WORD_63 : Word;   // F1009- F1024
   END_VAR
BEGIN
END_DATA_BLOCK

DATA_BLOCK "BM_MLT_GAP_SEARCH_DB"   // DB304
{ S7_Optimized_Access := 'FALSE' }
VERSION : 0.0
// stored: InstanceOfName BM_MLT_GAP_SEARCH
"BM_MLT_GAP_SEARCH"
BEGIN
END_DATA_BLOCK

DATA_BLOCK "BM_SEED_REF_POS_DB"   // DB305
{ S7_Optimized_Access := 'FALSE' }
VERSION : 0.0
// stored: InstanceOfName BM_SEED_REF_POS
"BM_SEED_REF_POS"
BEGIN
END_DATA_BLOCK

DATA_BLOCK "PM_MDI_DB"   // DB400
{ S7_Optimized_Access := 'FALSE' }
VERSION : 0.0
// stored: InstanceOfName PM_MDI
"PM_MDI"
BEGIN
END_DATA_BLOCK

DATA_BLOCK "PM_MDO_DB"   // DB401
{ S7_Optimized_Access := 'FALSE' }
VERSION : 0.0
// stored: InstanceOfName PM_MDO
"PM_MDO"
BEGIN
END_DATA_BLOCK

DATA_BLOCK "PM_MAI_DB"   // DB402
{ S7_Optimized_Access := 'FALSE' }
VERSION : 0.0
// stored: InstanceOfName PM_MAI
"PM_MAI"
BEGIN
END_DATA_BLOCK

DATA_BLOCK "PM_MAO_DB"   // DB403
{ S7_Optimized_Access := 'FALSE' }
VERSION : 0.0
// stored: InstanceOfName PM_MAO
"PM_MAO"
BEGIN
END_DATA_BLOCK

DATA_BLOCK "PM_INI_DI_DB"   // DB404
{ S7_Optimized_Access := 'FALSE' }
VERSION : 0.0
// stored: InstanceOfName PM_INI_DI
"PM_INI_DI"
BEGIN
END_DATA_BLOCK

DATA_BLOCK "PM_INI_AI_DB"   // DB405
{ S7_Optimized_Access := 'FALSE' }
VERSION : 0.0
// stored: InstanceOfName PM_INI_AI
"PM_INI_AI"
BEGIN
END_DATA_BLOCK

DATA_BLOCK "MDI"   // DB410
{ S7_Optimized_Access := 'FALSE' }
VERSION : 0.0
// --------------------------------------------------------------------------------
// program:             MDI
// description :        automatically generated MDI
// name:                hp
// date        :        03.02.2021
// 
// revision:
// name:
// date:
//                     (c)CGS
// --------------------------------------------------------------------------------
   VAR
      CB_FLT_DC24V_K2 : Bool;   // HDI def M 72.0: fault circuit breakers DC 24V 1=OK
      CB_FLT_AC400V_K2 : Bool;   // HDI def M 72.1: fault circuit breakers AC 400V 1=OK
      SPARE_16_2 : Bool;   // HDI def M 72.4: spare digital input
      CB_FLT_AC230V : Bool;   // HDI def M 72.3: fault circuit breakers AC 230V 1=OK
      SPARE_16_4 : Bool;   // HDI def M 72.4: spare digital input
      SPARE_16_5 : Bool;   // HDI def M 72.5: spare digital input
      SPARE_16_6 : Bool;   // HDI def M 72.6: spare digital input
      SPARE_16_7 : Bool;   // HDI def M 72.7: spare digital input
      SPARE_17_0 : Bool;   // HDI def M 73.0: spare digital input
      UPS_24V_ALM : Bool;   // HDI def M 73.1: alarm dc-usv
      UPS_24V_NRM : Bool;   // HDI def M 73.2: main line ready buffered dc-usv
      EMO : Bool;   // HDI def M 73.3: Emergency off (1=ok)
      EMS : Bool;   // HDI def M 73.4: Emergency stop handling drives (1=ok)
      SPARE_17_5 : Bool;   // HDI def M 73.5: spare digital input
      SPARE_17_6 : Bool;   // HDI def M 73.6: spare digital input
      SPARE_17_7 : Bool;   // HDI def M 73.7: spare digital input
      P1_WRN : Bool;   // HDI def M 74.0: pump unit (P1) warning
      P1_FLT : Bool;   // HDI def M 74.1: pump unit (P1) error
      P1_IS_ON : Bool;   // HDI def M 74.2: pump unit (P1) running
      P1_WD : Bool;   // HDI def M 74.3: pump unit (P1) watchdog
      FIL_APS : Bool;   // HDI def M 74.4: pressure filter 1000 mbar
      MON_TMP_P2 : Bool;   // HDI def M 74.5: temperature monitoring P2
      MON_TMP_P1 : Bool;   // HDI def M 74.6: temperature monitoring P1
      SPARE_18_7 : Bool;   // HDI def M 74.7: spare digital input
      FCH_LFT_SDL_NUT : Bool;   // HDI def M 88.0: safety limit switch furnace chamber lift spindle nut
      LS_FCH_LFT_DN : Bool;   // HDI def M 88.1: limit switch furnace chamber lift down
      LS_FCH_HOOK_WORK : Bool;   // HDI def M 88.2: limit switch furnace chamber hook in working position
      LS_FCH_HOOK_HOME : Bool;   // HDI def M 88.3: limit switch furnace chamber hook in home position
      LS_TEC_FLG_DN : Bool;   // HDI def M 88.4: limit switch technolgy flange down
      TEC_FLG_SDL_NUT : Bool;   // HDI def M 88.5: safety limit switch technolgy flange lift spindle nut
      LS_V11_COV_OP : Bool;   // HDI def M 88.6: Cover V11 opened (isolation valve feeder)
      LS_V11_COV_CL : Bool;   // HDI def M 88.7: Cover V11 closed (isolation valve feeder)
      GCH_APS : Bool;   // HDI def M 89.0: pressure gate chamber 1000 mbar
      FCH_APS : Bool;   // HDI def M 89.1: pressure furnace chamber 1000 mbar
      FDR_APS : Bool;   // HDI def M 89.2: pressure feeder 1000 mbar
      FIL_2_APS : Bool;   // HDI def M 89.3: atmospheric pressure filter 2
      SPARE_33_4 : Bool;   // HDI def M 89.4: spare
      SPARE_33_5 : Bool;   // HDI def M 89.5: spare
      LS_V2_1_OP : Bool;   // HDI def M 89.6: valve position v2.1 fce chamber
      LS_V2_1_CL : Bool;   // HDI def M 89.7: valve position v2.1 fce chamber
      CB_FLT_AC400V_K5 : Bool;   // HDI def M 90.0: fault circuit breakers AC 400V +K5 1=OK
      CB_FLT_DC24V_K5 : Bool;   // HDI def M 90.1: fault circuit breakers DC 24V +K5 1=OK
      LS_MAG_LFT_UP : Bool;   // HDI def M 90.2: limit switch magnet lift up
      LS_MAG_LFT_DN : Bool;   // HDI def M 90.3: limit switch magnet lift down
      SLS_MAG_LFT : Bool;   // HDI def M 90.4: Safety limit switch magnet lift
      MAG_LFT_SDL_NUT1 : Bool;   // HDI def M 90.5: safety limit switch magnet lift spindle nut 1
      MAG_LFT_SDL_NUT2 : Bool;   // HDI def M 90.6: safety limit switch magnet lift spindle nut 2
      MAG_LFT_SDL_NUT3 : Bool;   // HDI def M 90.7: safety limit switch magnet lift spindle nut 3
      OIL_LVL_CR_SFT : Bool;   // HDI def M 91.0: Crucible shaft min. oil level
      LS_V1_OP : Bool;   // HDI def M 91.1: V1 opened
      LS_V1_CL : Bool;   // HDI def M 91.2: V1 closed
      MP_ENB_K5 : Bool;   // HDI def M 91.3: Mobile panel agree button +K5
      SLS_TEC_FLG_LFT : Bool;   // HDI def M 91.4: Safety limit switch technolgy flange lift
      SLS_FCH_LFT : Bool;   // HDI def M 91.5: Safety limit switch furnace chamber lift
      COMP_AIR_OK : Bool;   // HDI def M 91.6: pressure switch compressed air ok
      COMP_AIR_2_OK : Bool;   // HDI def M 91.7: pressure switch compressed air 2 (ACC) ok
      LS_V1_1_CL : Bool;   // HDI def M 105.0: limit switch valve v1.1 closed
      LS_V1_1_OP : Bool;   // HDI def M 105.1: limit switch valve v1.1 opened
      LS_V3_4_OP : Bool;   // HDI def M 105.2: limit switch valve v3.4 opened
      LS_V3_4_CL : Bool;   // HDI def M 105.3: limit switch valve v3.4 closed
      LS_V3_3_OP : Bool;   // HDI def M 105.4: limit switch valve v3.3 opened
      LS_V3_3_CL : Bool;   // HDI def M 105.5: limit switch valve v3.3 closed
      LS_V2_11_OP : Bool;   // HDI def M 105.6: limit switch valve v2.11 opened
      LS_V2_11_CL : Bool;   // HDI def M 105.7: limit switch valve v2.11 closed
      ACC_FCH_OV_PRS_1 : Bool;   // HDI def M 92.0: ACC furnace overpressure 1
      ACC_FCH_OV_PRS_2 : Bool;   // HDI def M 92.1: ACC furnace overpressure 2
      SPARE_48_2 : Bool;   // HDI def M 92.2: ACC spare
      ACC_WTR_FLW_OUT_OK : Bool;   // HDI def M 92.3: ACC output waterflow ok
      ACC_WTR_FLW_IN_OK : Bool;   // HDI def M 92.4: ACC input waterflow ok
      ACC_WTR_TMP_OUT_OK : Bool;   // HDI def M 92.5: ACC output watertemp. Ok
      OV_PRS_1_FLT : Bool;   // HDI def M 92.6: ACC overpressure 1 error/fault
      OV_PRS_2_FLT : Bool;   // HDI def M 92.7: ACC overpressure 2 error/fault
      ACC_SC_WTR_OK : Bool;   // HDI def M 93.0: ACC safety circuit
      ACC_SC_WTR_ATV : Bool;   // HDI def M 93.1: ACC safety circuit
      ACC_SC_HTR_OK : Bool;   // HDI def M 93.2: ACC safety circuit
      ACC_SC_HTR_ATV : Bool;   // HDI def M 93.3: ACC safety circuit
      ACC_KEY_RST : Bool;   // HDI def M 93.4: ACC reset key
      ACC_CB_FLT_DC24V : Bool;   // HDI def M 93.5: ACC 24V circuit breaker ok
      ACC_UPS_24V_ALM : Bool;   // HDI def M 93.6: ACC UPS OK Normal
      ACC_UPS_24V_NRM : Bool;   // HDI def M 93.7: ACC UPS Alarm
      DPH_RPT_DET_OK : Bool;   // HDI def M 94.0: ACC Diaphraghm rupture detector OK
      ACC_CB_FLT_AC230V : Bool;   // HDI def M 94.1: Fault circuit breakers AC 230V
      SPARE_90_2 : Bool;   // HDI def M 94.2: ACC spare
      SPARE_90_3 : Bool;   // HDI def M 94.3: ACC spare
      SPARE_90_4 : Bool;   // HDI def M 94.4: ACC spare
      SPARE_90_5 : Bool;   // HDI def M 94.5: ACC spare
      SPARE_90_6 : Bool;   // HDI def M 94.6: ACC spare
      SPARE_90_7 : Bool;   // HDI def M 94.7: ACC spare
      FU_P2_RDY : Bool;   // HDI def M 104.0: Frequency converter P2 ready/ no fault
      SPARE_144_1 : Bool;   // HDI def M 104.1: spare digital input
      SPARE_144_2 : Bool;   // HDI def M 104.2: spare digital input
      SPARE_144_3 : Bool;   // HDI def M 104.3: spare digital input
      SPARE_144_4 : Bool;   // HDI def M 104.4: spare digital input
      SPARE_144_5 : Bool;   // HDI def M 104.5: spare digital input
      SPARE_144_6 : Bool;   // HDI def M 104.6: spare digital input
      SPARE_144_7 : Bool;   // HDI def M 104.7: spare digital input
      LS_GCH_UP : Bool;   // HDI def M 95.0: limit switch gate chamber in upper position
      LS_GCH_DN : Bool;   // HDI def M 95.1: limit switch gate chamber in lower position
      LS_GCH_SW_IN : Bool;   // HDI def M 95.2: limit switch gate chamber swivelled in
      LS_GCH_SW_CLN : Bool;   // HDI def M 95.3: limit switch gate chamber swivelled in cleaning pos
      LS_GCH_SW_OUT : Bool;   // HDI def M 95.4: limit switch gate chamber swivelled out
      LS_GCH_SW_LOCK : Bool;   // HDI def M 95.5: limit switch gate chamber swivel locked
      SLS_GCH_LFT : Bool;   // HDI def M 95.6: Safety limit switch gate chamber lift
      LS_TCH_UP : Bool;   // HDI def M 95.7: limit switch top chamber in upper position
      LS_TCH_DN : Bool;   // HDI def M 96.0: limit switch top chamber in lower position
      LS_TCH_SW_IN : Bool;   // HDI def M 96.1: limit switch top chamber swivelled in
      LS_TCH_SW_CLN : Bool;   // HDI def M 96.2: limit switch top chamber swivelled in cleaning pos
      LS_TCH_SW_OUT : Bool;   // HDI def M 96.3: limit switch top chamber swivelled out
      LS_TCH_SW_LOCK : Bool;   // HDI def M 96.4: limit switch top chamber swivel locked
      LS_TCH_TILT_0 : Bool;   // HDI def M 96.5: limit switch top chamber tilt 0?horizental
      LS_TCH_TILT_30 : Bool;   // HDI def M 96.6: limit switch top chamber tilt 30?Cleaning position
      KEY_XT_LFT_SRV : Bool;   // HDI def M 96.7: Key switch service mode crystal lift
      LS_V7_UP : Bool;   // HDI def M 97.0: limit switch gate valve V7 in upper position
      LS_V7_DN : Bool;   // HDI def M 97.1: limit switch gate valve V7 in lower position
      LS_V7_SW_IN : Bool;   // HDI def M 97.2: limit switch gate valve V7 swiveled in
      LS_V7_SW_OUT : Bool;   // HDI def M 97.3: limit switch gate valve V7 swiveled out
      LS_V7_FLP_OP : Bool;   // HDI def M 97.4: limit switch gate valve V7 flap open
      LS_V7_CLN_POS : Bool;   // HDI def M 97.5: limit switch gate valve V7 in cleaning position
      LS_GCH_BEL_UP : Bool;   // HDI def M 97.6: limit switch gate chamber bellow in upper position
      LS_GCH_BEL_DN : Bool;   // HDI def M 97.7: limit switch gate chamber bellow in lower position
      LS_XT_SLID_BW : Bool;   // HDI def M 98.0: limit switch crystal handling slider in home position
      LS_XT_SLID_FW : Bool;   // HDI def M 98.1: limit switch crystal handling slider in work position
      LS_XT_SLID_MID : Bool;   // HDI def M 98.2: limit switch crystal handling slider in middle position
      LS_XT_CLP_CON : Bool;   // HDI def M 98.3: limit switch crystal handling clamps connected
      LS_XT_TILT_90 : Bool;   // HDI def M 98.4: limit switch crystal handling tilt in 90?
      LS_XT_TILT_75 : Bool;   // HDI def M 98.5: limit switch crystal handling tilt in 75?
      LS_UP_XT_CLP_FLT : Bool;   // HDI def M 98.6: limit switch upper crystal clamp fault
      SPARE_275_7 : Bool;   // HDI def M 98.7: spare digital input
      LS_UP_XT_CLP_OP : Bool;   // HDI def M 99.0: limit switch upper crystal clamp open
      LS_UP_XT_CLP_CL : Bool;   // HDI def M 99.1: limit switch upper crystal clamp closed
      LS_UP_XT_CLP_SAVE : Bool;   // HDI def M 99.2: limit switch upper crystal clamp save
      LS_UP_XT_CLP_PLATE : Bool;   // HDI def M 99.3: limit switch upper crystal clamp plate
      LS_LO_XT_CLP_FLT : Bool;   // HDI def M 99.4: limit switch lower crystal clamp fault
      LS_LO_XT_CLP_OP : Bool;   // HDI def M 99.5: limit switch lower crystal clamp open
      LS_LO_XT_CLP_CL : Bool;   // HDI def M 99.6: limit switch lower crystal clamp closed
      LS_LO_XT_CLP_SAVE : Bool;   // HDI def M 99.7: limit switch lower crystal clamp save
      LS_LO_XT_CLP_PLATE : Bool;   // HDI def M 100.0: limit switch upper crystal clamp plate
      LS_HOI_TOOL_INST : Bool;   // HDI def M 100.1: limit switch HOI tool installed
      XT_DRP_OUT_PRT_1_CL : Bool;   // HDI def M 100.2: crystal drop out protection 1 closed (upper left side)
      XT_DRP_OUT_PRT_1_OP : Bool;   // HDI def M 100.3: crystal drop out protection 1 opened (upper left side)
      XT_DRP_OUT_PRT_2_CL : Bool;   // HDI def M 100.4: crystal drop out protection 2 closed (upper right side)
      XT_DRP_OUT_PRT_2_OP : Bool;   // HDI def M 100.5: crystal drop out protection 2 opened (upper right side)
      CB_FLT_AC400V_K8 : Bool;   // HDI def M 100.6: fault circuit breakers AC 400V 1=OK
      CB_FLT_DC24V_K8 : Bool;   // HDI def M 100.7: fault circuit breakers DC 24V 1=OK
      XT_DRP_OUT_PRT_3_CL : Bool;   // HDI def M 101.0: crystal drop out protection 3 closed (lower left side)
      XT_DRP_OUT_PRT_3_OP : Bool;   // HDI def M 101.1: crystal drop out protection 3 opened (lower left side)
      XT_DRP_OUT_PRT_4_CL : Bool;   // HDI def M 101.2: crystal drop out protection 4 closed (lower right side)
      XT_DRP_OUT_PRT_4_OP : Bool;   // HDI def M 101.3: crystal drop out protection 4 opened (lower right side)
      LS_XT_HDL_SW_UNLOCK : Bool;   // HDI def M 101.4: limit switch crystal handling swivel unlocked
      LS_XT_HDL_SW_LOCK : Bool;   // HDI def M 101.5: limit switch crystal handling swivel locked 145?
      LS_GCH_DOOR_OP : Bool;   // HDI def M 101.6: limit switch gate chamber door opened
      LS_GCH_DOOR_CL : Bool;   // HDI def M 101.7: limit switch gate chamber door closed
      MCC_CONTACT_XT : Bool;   // HDI def M 102.0: seed contact detection (xt isolated)
      OIL_LVL_XT_SFT : Bool;   // HDI def M 102.1: Crystal shaft min. oil level
      LS_XT_SFT_SRV_POS : Bool;   // HDI def M 102.2: limit switch crystal shaft service position
      LS_XT_TOP_POS : Bool;   // HDI def M 102.3: limit switch crystal shaft in top position
      SLS_TCH_LFT : Bool;   // HDI def M 102.4: Safety limit switch top chamber lift
      XT_ROT_CAM_TRG : Bool;   // HDI def M 102.5: limit switch xtal rotation camera trigger
      MP_ENB_K8 : Bool;   // HDI def M 102.6: Mobile panel agree button +K8
      MP_ENB_K9 : Bool;   // HDI def M 102.7: Mobile panel agree button +K9
      LS_V3_OP : Bool;   // HDI def M 103.0: valve position V3 open
      LS_V3_CL : Bool;   // HDI def M 103.1: Valve position V3 closed
      FDR_LS_V3_2_OP : Bool;   // HDI def M 103.2: valve position V3_2 open
      FDR_LS_V3_2_CL : Bool;   // HDI def M 103.3: Valve position V3_2 closed
      LSR_SEN_OBJ_DET : Bool;   // HDI def M 103.4: spare digital input
      SPARE_280_5 : Bool;   // HDI def M 103.5: spare digital input
      SPARE_280_6 : Bool;   // HDI def M 103.6: spare digital input
      SPARE_280_7 : Bool;   // HDI def M 103.7: spare digital input
      LS_V11_OP : Bool;   // HDI def M 89.3: V 11 open (isolation valve feeder)
      LS_V11_CL : Bool;   // HDI def M 89.4: V 11 closed (isolation valve feeder)
      FDR_HOP_CON : Bool;   // HDI def M 89.5: hopper connected to feeder
   END_VAR
BEGIN
END_DATA_BLOCK

DATA_BLOCK "MDO"   // DB411
{ S7_Optimized_Access := 'FALSE' }
VERSION : 0.0
// --------------------------------------------------------------------------------
// program:             MDO
// description :        automatically generated MDO
// name:                hp
// date        :        03.02.2021
// 
// revision:
// name:
// date:
//                     (c)CGS
// --------------------------------------------------------------------------------
   VAR
      HOR_OPP_K2 : Bool;   // HDO def M 136.0: Horn +K2
      LMP_RD_K2 : Bool;   // HDO def M 136.1: Lamp red +K2
      LMP_YE_K2 : Bool;   // HDO def M 136.2: Lamp yellow +K2
      LMP_GN_K2 : Bool;   // HDO def M 136.3: Lamp green +K2
      LMP_BU_K2 : Bool;   // HDO def M 136.4: Lamp blue +K2
      HOR_MAG_ACTIVE : Bool;   // HDO def M 136.5: Horn magnet active( Lift)
      LMP_MAG_ACTIVE : Bool;   // HDO def M 136.6: Lamp magnet active( Lift+ Field on)
      SPARE_16_7 : Bool;   // HDO def M 136.7: spare digital output
      P1_ON : Bool;   // HDO def M 137.0: Vacuum pump 1 on (furnace chamber)
      P3_ON : Bool;   // HDO def M 137.1: Vacuum pump 3 on (gate chamber)
      P2_ON : Bool;   // HDO def M 137.2: Vacuum pump 2 on (roots furnace chamber)
      P1_SEAL_GAS : Bool;   // HDO def M 137.3: Vacuum pump 1 seal gas on
      P3_SEAL_GAS : Bool;   // HDO def M 137.4: Vacuum pump 3 seal gas on
      HTR_PWR_ON : Bool;   // HDO def M 137.4: Heater power supply on
      V10 : Bool;   // HDO def M 137.6: Vacuum pump 1 secuvac valve V10 on
      MON_TMP_P2_RES : Bool;   // HDO def M 137.7: temperature monitoring pump 2 reset
      SPARE_18_0 : Bool;   // HDO def M 138.0: spare digital output
      SPARE_18_1 : Bool;   // HDO def M 138.1: spare digital output
      SPARE_18_2 : Bool;   // HDO def M 138.2: spare digital output
      SPARE_18_3 : Bool;   // HDO def M 138.3: spare digital output
      SPARE_18_4 : Bool;   // HDO def M 138.4: spare digital output
      SPARE_18_5 : Bool;   // HDO def M 138.5: spare digital output
      SPARE_18_6 : Bool;   // HDO def M 138.6: spare digital output
      SPARE_18_7 : Bool;   // HDO def M 138.7: spare digital output
      V1_OP : Bool;   // HDO def M 142.0: V1 open
      V1_CL : Bool;   // HDO def M 142.1: V1 close
      SPARE_32_2 : Bool;   // HDO def M 142.2: spare digital output
      SPARE_32_3 : Bool;   // HDO def M 142.3: spare digital output
      SPARE_32_4 : Bool;   // HDO def M 142.4: spare digital output
      CR_ROT_ENB : Bool;   // HDO def M 142.5: controller enable crucible rotation
      CR_LFT_ENB : Bool;   // HDO def M 142.6: controller enable crucible lift
      FU_FCB_HDL_ON : Bool;   // HDO def M 142.7: Frequency converter FCB handling on
      TEC_FLG_LFT_ENB : Bool;   // HDO def M 143.0: controller enable techn chamber lift
      FCH_LFT_ENB : Bool;   // HDO def M 143.1: controller enable lower chamber parts lift
      MAG_LFT_UP : Bool;   // HDO def M 143.2: Magnet lift drive upwards
      MAG_LFT_DN : Bool;   // HDO def M 143.3: Magnet lift drive downwards
      BRK_MAG_LFT : Bool;   // HDO def M 143.4: Brake magnet lift
      SPARE_33_5 : Bool;   // HDO def M 143.5: spare digital output
      SPARE_33_6 : Bool;   // HDO def M 143.6: spare digital output
      SPARE_33_7 : Bool;   // HDO def M 143.7: spare digital output
      V1_1_OP : Bool;   // HDO def M 144.0: V1.1 open
      V1_1_CL : Bool;   // HDO def M 144.1: V1.1 close
      SPARE_34_2 : Bool;   // HDO def M 144.2: spare digital output
      SPARE_34_3 : Bool;   // HDO def M 144.3: spare digital output
      SPARE_34_4 : Bool;   // HDO def M 144.4: spare digital output
      SPARE_34_5 : Bool;   // HDO def M 144.5: spare digital output
      SPARE_34_6 : Bool;   // HDO def M 144.6: spare digital output
      SPARE_34_7 : Bool;   // HDO def M 144.7: spare digital output
      ACC_SC_HTR_STR : Bool;   // HDO def M 146.0: ACC Heizung START
      ACC_SC_HTR_RST : Bool;   // HDO def M 146.1: ACC Heizung RESET
      ACC_SC_WTR_STR : Bool;   // HDO def M 146.2: ACC K黨lwasser START
      ACC_SC_WTR_RST : Bool;   // HDO def M 146.3: ACC K黨lwasser RESET
      ACC_ALM_LT_1 : Bool;   // HDO def M 146.4: ACC Blitzlicht Kasten
      ACC_ALM_SND_1 : Bool;   // HDO def M 146.5: ACC Sirene Kasten
      ACC_ALM_LT_2 : Bool;   // HDO def M 146.6: ACC Blitzlicht Bedienpult
      ACC_ALM_SND_2 : Bool;   // HDO def M 146.7: ACC Sirene Bedienpult
      FCH_HOOK_HOME : Bool;   // HDO def M 150.0: Valve block lower furnace chamber hook unlocking
      FCH_HOOK_WORK : Bool;   // HDO def M 150.1: Valve block lower furnace chamber hook locking
      UP_FCH_SW_BRK : Bool;   // HDO def M 150.2: Valve block upper chamber swivel release brake
      LO_FCH_SW_BRK : Bool;   // HDO def M 150.3: Valve block lower chamber swivel release brake
      TEC_FLG_SW_BRK : Bool;   // HDO def M 150.4: Valve block tech. flange swivel release brake
      V25 : Bool;   // HDO def M 150.5: Valve block argon inlet pressure storage tank, V25 open
      V2_1 : Bool;   // HDO def M 150.6: Valve block vacuum valve, V2.1 open
      V21 : Bool;   // HDO def M 150.7: Valve block air valve vacuum pipe, V21+V21.1 open
      V19 : Bool;   // HDO def M 151.0: Valve block extraktion valve filter, V19 open
      V20 : Bool;   // HDO def M 151.1: Valve block air valve filter, V20 open
      V22 : Bool;   // HDO def M 151.2: Valve block argon valve filter, V22 open
      V9_2 : Bool;   // HDO def M 151.3: Valve block ventiliation valve vaccum line gate, V9_2
      V22_1 : Bool;   // HDO def M 151.4: Valve block argon valve bypass filter, V22.1 open
      V3_4 : Bool;   // HDO def M 151.5: Valve block vacuum valve, V3.4 open
      V3_3 : Bool;   // HDO def M 151.6: Valve block vacuum valve, V3.3 open
      V2_11 : Bool;   // HDO def M 151.7: Valve block vacuum valve, V2.11 open
      P2_FU_ON : Bool;   // HDO def M 152.0: Frequency converter P2 start
      P2_FU_RES : Bool;   // HDO def M 152.1: Frequency converter P2 fault reset
      SPARE_144_2 : Bool;   // HDO def M 152.2: spare digital output
      SPARE_144_3 : Bool;   // HDO def M 152.3: spare digital output
      SPARE_144_4 : Bool;   // HDO def M 152.4: spare digital output
      SPARE_144_5 : Bool;   // HDO def M 152.5: spare digital output
      SPARE_144_6 : Bool;   // HDO def M 152.6: spare digital output
      SPARE_144_7 : Bool;   // HDO def M 152.7: spare digital output
      V4 : Bool;   // HDO def M 150.0: Valve block V4 valve argon gas inlet (gate chamber)
      V5 : Bool;   // HDO def M 150.1: Valve block V5 valve argon gas inlet controlled (gch)
      V6 : Bool;   // HDO def M 150.2: Valve block V6 valve argon gas inlet controlled (Fch)
      V3 : Bool;   // HDO def M 150.3: Valve block V3 vacuum valve (gate chamber)
      V3_2 : Bool;   // HDO def M 150.4: Valve block V3.2 vacuum valve feeder
      V24 : Bool;   // HDO def M 150.5: Valve block V24 valve argon gas inlet feeder
      XT_DRP_OUT_PRT_CL : Bool;   // HDO def M 150.6: Valve block close crystal drop out protection
      XT_DRP_OUT_PRT_OP : Bool;   // HDO def M 150.7: Valve block open crystal drop out protection
      TCH_SW_LOCK : Bool;   // HDO def M 151.0: Valve block top chamber swivel lock close
      TCH_SW_UNLOCK : Bool;   // HDO def M 151.1: Valve block top chamber swivel lock open
      GCH_SW_LOCK : Bool;   // HDO def M 151.2: Valve block gate chamber swivel lock close
      GCH_SW_UNLOCK : Bool;   // HDO def M 151.3: Valve block gate chamber swivel lock open
      XT_HDL_SW_LOCK : Bool;   // HDO def M 151.4: Valve block xtal handling swivel lock close (145?
      XT_HDL_SW_UNLOCK : Bool;   // HDO def M 151.5: Valve block xtal handling swivel lock open (145?
      FDR_V11_OP : Bool;   // HDO def M 151.6: Valve block open V11 (isolation valve feeder)
      FDR_V11_CL : Bool;   // HDO def M 151.7: Valve block close V11 (isolation valve feeder)
      FDR_V11_CVR_OP : Bool;   // HDO def M 152.0: Valve block open cover V11 (isolation valve feeder)
      FDR_V11_CVR_CL : Bool;   // HDO def M 152.1: Valve block close cover V11 (isolation valve feeder)
      SPARE_226_2 : Bool;   // HDO def M 152.2: Valve block spare output
      SPARE_226_3 : Bool;   // HDO def M 152.3: Valve block spare output
      SPARE_226_4 : Bool;   // HDO def M 152.4: Valve block spare output
      SPARE_226_5 : Bool;   // HDO def M 152.5: Valve block spare output
      SPARE_226_6 : Bool;   // HDO def M 152.6: Valve block spare output
      SPARE_226_7 : Bool;   // HDO def M 152.7: Valve block spare output
      HOR_OPP_K8 : Bool;   // HDO def M 160.0: Horn +K8
      LMP_RD_K8 : Bool;   // HDO def M 160.1: Lamp red +K8
      LMP_YE_K8 : Bool;   // HDO def M 160.2: Lamp yellow +K8
      LMP_GN_K8 : Bool;   // HDO def M 160.3: Lamp green +K8
      LMP_BU_K8 : Bool;   // HDO def M 160.4: Lamp blue +K8
      XT_ROT_ENB : Bool;   // HDO def M 160.5: controller enable crystal rotation
      XT_LFT_ENB : Bool;   // HDO def M 160.6: controller enable crystal lift
      XT_HDL_LFT_ENB : Bool;   // HDO def M 160.7: controller enable crystal handling lift
      XT_HDL_SW_ENB : Bool;   // HDO def M 161.0: controller enable crystal handling swivel
      FU_GCB_HDL_ON : Bool;   // HDO def M 161.1: Frequency converter GCB handling on
      LSR_SEN_PWR_ON : Bool;   // HDO def M 161.2: supply voltage for laser sensor on
      SPARE_273_3 : Bool;   // HDO def M 161.3: spare digital output
      SPARE_273_4 : Bool;   // HDO def M 161.4: spare digital output
      SPARE_273_5 : Bool;   // HDO def M 161.5: spare digital output
      XT_HDL_SLID_FW : Bool;   // HDO def M 161.6: Motor crystal handling slider forwards
      XT_HDL_SLID_BW : Bool;   // HDO def M 161.7: Motor crystal handling slider backwards
      XT_CLP_TILT_BW : Bool;   // HDO def M 163.0: Motor crystal clamp tilt backwards
      XT_CLP_TILT_FW : Bool;   // HDO def M 163.1: Motor crystal clamp tilt forwards (75?
      XT_CLP_TILT_BRK : Bool;   // HDO def M 163.2: Motor crystal clamp tilt brake
      XT_CLP_ABV_OP : Bool;   // HDO def M 163.3: Motor crystal clamp above open
      XT_CLP_ABV_CL : Bool;   // HDO def M 163.4: Motor crystal clamp above close
      XT_CLP_ABV_BRK : Bool;   // HDO def M 163.5: Brake crystal clamp above
      XT_CLP_ABV_RST : Bool;   // HDO def M 163.6: Reset controller crystal clamp above
      GCH_LFT_ENB : Bool;   // HDO def M 163.7: controller enable gate chamber lift
      XT_CLP_BLW_OP : Bool;   // HDO def M 164.0: Motor crystal clamp below open
      XT_CLP_BLW_CL : Bool;   // HDO def M 164.1: Motor crystal clamp below close
      XT_CLP_BLW_BRK : Bool;   // HDO def M 164.2: Brake crystal clamp below
      XT_CLP_BLW_RST : Bool;   // HDO def M 164.3: Reset controller crystal clamp below
      MCC_TEST_XT : Bool;   // HDO def M 164.4: seed contact detection test output ( xt isolated)
      MCC_ENB_XT : Bool;   // HDO def M 164.5: seed contact detection enable output (xt isolated)
      TCH_LFT_ENB : Bool;   // HDO def M 164.6: controller enable top chamber lift
      TCH_TILT_ENB : Bool;   // HDO def M 164.7: controller enable top chamber tilt
      GTE_V_LFT_ENB : Bool;   // HDO def M 165.0: controller enable gate valve lift
      GTE_V_SW_ENB : Bool;   // HDO def M 165.1: controller enable gate valve swivel
      BEL_LFT_ENB : Bool;   // HDO def M 165.2: controller enable gate bellow lift
      HOR_OPP_K9 : Bool;   // HDO def M 165.3: Horn +K9
      LMP_RD_K9 : Bool;   // HDO def M 165.4: Lamp red +K9
      LMP_YE_K9 : Bool;   // HDO def M 165.5: Lamp yellow +K9
      LMP_GN_K9 : Bool;   // HDO def M 165.6: Lamp green +K9
      LMP_BU_K9 : Bool;   // HDO def M 165.7: Lamp blue +K9
   END_VAR
BEGIN
END_DATA_BLOCK

DATA_BLOCK "MAI"   // DB412
{ S7_Optimized_Access := 'FALSE' }
VERSION : 0.0
// --------------------------------------------------------------------------------
// program:             MAI
// description :        automatically generated MAI
// name:                hp
// date        :        03.02.2021
// 
// revision:
// name:
// date:
//                     (c)CGS
// --------------------------------------------------------------------------------
   VAR
      TRV_ACT_POS : Real;   // HAI def MW 192: actual throttle valve position
      TRV_ACT_POS_1 : Real;   // HAI def MW 194: actual throttle valve 1.1 position
      TRV_PRS_FIL_1 : Real;   // HAI def MW 204: actual pressure value main filter
      TRV_PRS_FIL_2 : Real;   // HAI def MW 206: actual pressure value bypass filter
      PYR_ACT_HTR_1_TMP : Real;   // HAI def MW 250: actual temperature main heater
      ACT_PRS_AR_VSL : Real;   // HAI def MW 252: actual pressure argon storage tank
      SPARE_484 : Real;   // HAI def MW 254: spare analog output (4..20 mA)
      SPARE_486 : Real;   // HAI def MW 256: spare analog output (4..20 mA)
      PYR_ACT_MELT_TMP : Real;   // HAI def MW 280: actual temperature melt
      SPARE_1538 : Real;   // HAI def MW 282: spare analog output (4..20 mA)
      SPARE_1540 : Real;   // HAI def MW 284: spare analog output (4..20 mA)
      SPARE_1542 : Real;   // HAI def MW 286: spare analog output (4..20 mA)
      GCH_PCR_ACT_PRS : Real;   // HAI def MW 242: actual vacuum gauge gate chamber 5xe-4...1500 mbar
      FCH_PCR_ACT_PRS : Real;   // HAI def MW 200: actual vacuum gauge furnace chamber 5xe-4...1500 mbar
      FCH_BAR_ACT_PRS_100 : Real;   // HAI def MW 198: actual vacuum gauge furnace chamber 100 mbar
      ACC_WTR_TMP : Real;   // HAI def MW 258: ACC water temp.
      ACC_WTR_PRS_IN : Real;   // HAI def MW 260: ACC water pressure
      ACC_WTR_FLW_OUT : Real;   // HAI def MW 262: ACC waterflow output
      ACC_WTR_FLW_IN : Real;   // HAI def MW 264: ACC waterflow input
      ACC_WTR_SPL_PRS : Real;   // HAI def MW 266: ACC water supply inlet pressure
      ACC_SPARE_810 : Real;   // HAI def MW 268: ACC spare
      SPARE : Real;   // HAI def MW 270: spare
   END_VAR
BEGIN
END_DATA_BLOCK

DATA_BLOCK "MAO"   // DB413
{ S7_Optimized_Access := 'FALSE' }
VERSION : 0.0
// --------------------------------------------------------------------------------
// program:             MAO
// description :        automatically generated MAO
// name:                hp
// date        :        03.02.2021
// 
// revision:
// name:
// date:
//                     (c)CGS
// --------------------------------------------------------------------------------
   VAR
      TRV_SET_POS : Real;   // HAO def MW 300: setpoint throttle valve 1 position
      TRV_SET_POS_1 : Real;   // HAO def MW 302: setpoint throttle valve 1.1 position
      SPARE : Real;   // HAO def MW 304: spare
   END_VAR
BEGIN
END_DATA_BLOCK

DATA_BLOCK "HAI"   // DB414
{ S7_Optimized_Access := 'FALSE' }
VERSION : 0.0
// --------------------------------------------------------------------------------
// program:             HAI
// description :        automatically generated HAI
// name:                hp
// date        :        03.02.2021
// 
// revision:
// name:
// date:
//                     (c)CGS
// --------------------------------------------------------------------------------
   VAR
      TRV_ACT_POS : Real;   // HAI def MW 192: actual throttle valve position
      TRV_ACT_POS_1 : Real;   // HAI def MW 194: actual throttle valve 1.1 position
      TRV_PRS_FIL_1 : Real;   // HAI def MW 204: actual pressure value main filter
      TRV_PRS_FIL_2 : Real;   // HAI def MW 206: actual pressure value bypass filter
      PYR_ACT_HTR_1_TMP : Real;   // HAI def MW 250: actual temperature main heater
      ACT_PRS_AR_VSL : Real;   // HAI def MW 252: actual pressure argon storage tank
      SPARE_484 : Real;   // HAI def MW 254: spare analog output (4..20 mA)
      SPARE_486 : Real;   // HAI def MW 256: spare analog output (4..20 mA)
      PYR_ACT_MELT_TMP : Real;   // HAI def MW 280: actual temperature melt
      SPARE_1538 : Real;   // HAI def MW 282: spare analog output (4..20 mA)
      SPARE_1540 : Real;   // HAI def MW 284: spare analog output (4..20 mA)
      SPARE_1542 : Real;   // HAI def MW 286: spare analog output (4..20 mA)
      GCH_PCR_ACT_PRS : Real;   // HAI def MW 242: actual vacuum gauge gate chamber 5xe-4...1500 mbar
      FCH_PCR_ACT_PRS : Real;   // HAI def MW 200: actual vacuum gauge furnace chamber 5xe-4...1500 mbar
      FCH_BAR_ACT_PRS_100 : Real;   // HAI def MW 198: actual vacuum gauge furnace chamber 100 mbar
      ACC_WTR_TMP : Real;   // HAI def MW 258: ACC water temp.
      ACC_WTR_PRS_IN : Real;   // HAI def MW 260: ACC water pressure
      ACC_WTR_FLW_OUT : Real;   // HAI def MW 262: ACC waterflow output
      ACC_WTR_FLW_IN : Real;   // HAI def MW 264: ACC waterflow input
      ACC_WTR_SPL_PRS : Real;   // HAI def MW 266: ACC water supply inlet pressure
      ACC_SPARE_810 : Real;   // HAI def MW 268: ACC spare
      SPARE : Real;   // HAI def MW 270: spare
   END_VAR
BEGIN
END_DATA_BLOCK

DATA_BLOCK "HAO"   // DB415
{ S7_Optimized_Access := 'FALSE' }
VERSION : 0.0
// --------------------------------------------------------------------------------
// program:             HAO
// description :        automatically generated HAO
// name:                hp
// date        :        03.02.2021
// 
// revision:
// name:
// date:
//                     (c)CGS
// --------------------------------------------------------------------------------
   VAR
      TRV_SET_POS : Real;   // HAO def MW 300: setpoint throttle valve 1 position
      TRV_SET_POS_1 : Real;   // HAO def MW 302: setpoint throttle valve 1.1 position
      SPARE : Real;   // HAO def MW 304: spare
   END_VAR
BEGIN
END_DATA_BLOCK

DATA_BLOCK "BM_VAC_DB"   // DB500
{ S7_Optimized_Access := 'FALSE' }
VERSION : 0.0
// stored: InstanceOfName BM_VAC_MAIN
"BM_VAC_MAIN"
BEGIN
END_DATA_BLOCK

DATA_BLOCK "BM_FIL_CHG_DB"   // DB501
{ S7_Optimized_Access := 'FALSE' }
VERSION : 0.0
// stored: InstanceOfName BM_FIL_CHG
"BM_FIL_CHG"
BEGIN
END_DATA_BLOCK

DATA_BLOCK "PM_DI_DB"   // DB512
{ S7_Optimized_Access := 'FALSE' }
VERSION : 0.0
// stored: InstanceOfName PM_DI
"PM_DI"
BEGIN
END_DATA_BLOCK

DATA_BLOCK "PM_DO_DB"   // DB513
{ S7_Optimized_Access := 'FALSE' }
VERSION : 0.0
// stored: InstanceOfName PM_DO
"PM_DO"
BEGIN
END_DATA_BLOCK

DATA_BLOCK "PM_AI_DB"   // DB514
{ S7_Optimized_Access := 'FALSE' }
VERSION : 0.0
// stored: InstanceOfName PM_AI
"PM_AI"
BEGIN
END_DATA_BLOCK

DATA_BLOCK "PM_AO_DB"   // DB515
{ S7_Optimized_Access := 'FALSE' }
VERSION : 0.0
// stored: InstanceOfName PM_AO
"PM_AO"
BEGIN
END_DATA_BLOCK

DATA_BLOCK "PM"   // DB516
{ S7_Optimized_Access := 'FALSE' }
VERSION : 0.0
// --------------------------------------------------------------------------------
//     program     :    PM
//     description :    misc data for pm modules
//                            
//     name        :    G. Eibelsh鋟ser
//     date        :    29.07.2009
// 
//     revision    :
//     name        :
//     date        :    
//                     (c)PVATepla AG
//     --------------------------------------------------------------------------------
   VAR
      CTRL_DATA_DVC_DRV : Array[1..9] of Struct
         cw : Bool;
         ccw : Bool;
         stop : Bool;
         set_point : Real;
         cw_active : Bool;
         ccw_active : Bool;
         stop_active : Bool;
         actual : Real;
         fault : Bool;
      END_STRUCT;
      CTRL_DATA_DVC_DRV_OFF : Struct
         cw : Bool;
         ccw : Bool;
         stop : Bool := TRUE;
         set_point : Real;
         cw_active : Bool;
         ccw_active : Bool;
         stop_active : Bool;
         actual : Real;
         fault : Bool;
      END_STRUCT;
      CTRL_DATA_DVC_PS : Array[20..29] of Struct
         on : Bool;
         off : Bool;
         set_pwr : Real;
         set_cur : Real;
         on_active : Bool;
         off_active : Bool;
         msg : Word;   // description see below
         act_pwr : Real;
         act_cur : Real;
         act_vlt : Real;
         act_res : Real;
      END_STRUCT;
      CTRL_DATA_DVC_PS_OFF : Struct
         on : Bool;
         off : Bool := TRUE;
         set_pwr : Real;
         set_cur : Real;
         on_active : Bool;
         off_active : Bool;
         msg : Word;
         act_pwr : Real;
         act_cur : Real;
         act_vlt : Real;
         act_res : Real;
      END_STRUCT;
   END_VAR
BEGIN
END_DATA_BLOCK

DATA_BLOCK "PM_DEVICE_IRCON_R727"   // DB517
{ S7_Optimized_Access := 'FALSE' }
VERSION : 0.0
// --------------------------------------------------------------------------------
//     program     :    PM_DEVICE_IRCON_R727
//     description :    Characteristic curve of IRCON SPECIAL R727 infrared pyrometer
//                      signal :    output current in micro amps
//                      temp   :    temperature in degree C     
//     name        :    G. Eibelsh鋟ser
//     date        :    08.12.99
// 
//     revision    :
//     name        :
//     date        :    
//                     (c)CGS
//     --------------------------------------------------------------------------------
   VAR
      signal : Array[1..46] of Real;
      temp : Array[1..46] of Real;
   END_VAR
BEGIN
   signal[1] := 0.797666;
   signal[2] := 0.966433;
   signal[3] := 1.164348;
   signal[4] := 1.395282;
   signal[5] := 1.663451;
   signal[6] := 1.97343;
   signal[7] := 2.330167;
   signal[8] := 2.738991;
   signal[9] := 3.205624;
   signal[10] := 3.736185;
   signal[11] := 4.337204;
   signal[12] := 5.015621;
   signal[13] := 5.778796;
   signal[14] := 6.634507;
   signal[15] := 7.590959;
   signal[16] := 8.656778;
   signal[17] := 9.841014;
   signal[18] := 11.15314;
   signal[19] := 12.60304;
   signal[20] := 14.20103;
   signal[21] := 15.95781;
   signal[22] := 17.8845;
   signal[23] := 19.99261;
   signal[24] := 22.29404;
   signal[25] := 24.80106;
   signal[26] := 27.52631;
   signal[27] := 30.48278;
   signal[28] := 33.68381;
   signal[29] := 37.14306;
   signal[30] := 40.87452;
   signal[31] := 44.89248;
   signal[32] := 49.21149;
   signal[33] := 53.84642;
   signal[34] := 58.81236;
   signal[35] := 64.12466;
   signal[36] := 69.79888;
   signal[37] := 75.85081;
   signal[38] := 82.29642;
   signal[39] := 89.15183;
   signal[40] := 96.43338;
   signal[41] := 104.1575;
   signal[42] := 112.3407;
   signal[43] := 120.9998;
   signal[44] := 130.1515;
   signal[45] := 139.8126;
   signal[46] := 150.0;
   temp[1] := 1000.0;
   temp[2] := 1020.0;
   temp[3] := 1040.0;
   temp[4] := 1060.0;
   temp[5] := 1080.0;
   temp[6] := 1100.0;
   temp[7] := 1120.0;
   temp[8] := 1140.0;
   temp[9] := 1160.0;
   temp[10] := 1180.0;
   temp[11] := 1200.0;
   temp[12] := 1220.0;
   temp[13] := 1240.0;
   temp[14] := 1260.0;
   temp[15] := 1280.0;
   temp[16] := 1300.0;
   temp[17] := 1320.0;
   temp[18] := 1340.0;
   temp[19] := 1360.0;
   temp[20] := 1380.0;
   temp[21] := 1400.0;
   temp[22] := 1420.0;
   temp[23] := 1440.0;
   temp[24] := 1460.0;
   temp[25] := 1480.0;
   temp[26] := 1500.0;
   temp[27] := 1520.0;
   temp[28] := 1540.0;
   temp[29] := 1560.0;
   temp[30] := 1580.0;
   temp[31] := 1600.0;
   temp[32] := 1620.0;
   temp[33] := 1640.0;
   temp[34] := 1660.0;
   temp[35] := 1680.0;
   temp[36] := 1700.0;
   temp[37] := 1720.0;
   temp[38] := 1740.0;
   temp[39] := 1760.0;
   temp[40] := 1780.0;
   temp[41] := 1800.0;
   temp[42] := 1820.0;
   temp[43] := 1840.0;
   temp[44] := 1860.0;
   temp[45] := 1880.0;
   temp[46] := 1900.0;
END_DATA_BLOCK

DATA_BLOCK "PM_DEVICE_IRCON_11x20"   // DB518
{ S7_Optimized_Access := 'FALSE' }
VERSION : 0.0
// --------------------------------------------------------------------------------
//     program     :    PM_DEVICE_IRCON_11x20
//     description :    Characteristic curve of IRCON 11x20 infrared pyrometer
//                      signal :    output current in mV
//                      temp   :    temperature in degree C     
//     name        :    G. Eibelsh鋟ser
//     date        :    08.08.2000
// 
//     revision    :
//     name        :
//     date        :    
//                     (c)CGS
//     --------------------------------------------------------------------------------
   VAR
      signal : Array[1..46] of Real;
      temp : Array[1..46] of Real;
   END_VAR
BEGIN
   signal[1] := 2.625;
   signal[2] := 3.075;
   signal[3] := 3.5;
   signal[4] := 4.0;
   signal[5] := 4.55;
   signal[6] := 5.1;
   signal[7] := 5.7;
   signal[8] := 6.375;
   signal[9] := 7.125;
   signal[10] := 7.95;
   signal[11] := 8.8;
   signal[12] := 9.65;
   signal[13] := 10.7;
   signal[14] := 11.85;
   signal[15] := 13.05;
   signal[16] := 14.4;
   signal[17] := 15.75;
   signal[18] := 17.25;
   signal[19] := 19.0;
   signal[20] := 20.75;
   signal[21] := 22.75;
   signal[22] := 24.9;
   signal[23] := 27.0;
   signal[24] := 29.5;
   signal[25] := 32.0;
   signal[26] := 34.75;
   signal[27] := 37.5;
   signal[28] := 40.75;
   signal[29] := 44.0;
   signal[30] := 47.25;
   signal[31] := 50.0;
   temp[1] := 1300.0;
   temp[2] := 1320.0;
   temp[3] := 1340.0;
   temp[4] := 1360.0;
   temp[5] := 1380.0;
   temp[6] := 1400.0;
   temp[7] := 1420.0;
   temp[8] := 1440.0;
   temp[9] := 1460.0;
   temp[10] := 1480.0;
   temp[11] := 1500.0;
   temp[12] := 1520.0;
   temp[13] := 1540.0;
   temp[14] := 1560.0;
   temp[15] := 1580.0;
   temp[16] := 1600.0;
   temp[17] := 1620.0;
   temp[18] := 1640.0;
   temp[19] := 1660.0;
   temp[20] := 1680.0;
   temp[21] := 1700.0;
   temp[22] := 1720.0;
   temp[23] := 1740.0;
   temp[24] := 1760.0;
   temp[25] := 1780.0;
   temp[26] := 1800.0;
   temp[27] := 1820.0;
   temp[28] := 1840.0;
   temp[29] := 1860.0;
   temp[30] := 1880.0;
   temp[31] := 1900.0;
END_DATA_BLOCK

DATA_BLOCK "PM_GET_WGT_XT_CLP_DB"   // DB531
{ S7_Optimized_Access := 'FALSE' }
VERSION : 0.0
// stored: InstanceOfName PM_GET_WGT_XT_CLP
"PM_GET_WGT_XT_CLP"
BEGIN
END_DATA_BLOCK

DATA_BLOCK "CM_LOOP_PRS_DB"   // DB544
{ S7_Optimized_Access := 'FALSE' }
VERSION : 0.0
// stored: InstanceOfName CM_LOOP_PRS
"CM_LOOP_PRS"
BEGIN
END_DATA_BLOCK

DATA_BLOCK "CM_LOOP_DIA_DB"   // DB545
{ S7_Optimized_Access := 'FALSE' }
VERSION : 0.0
// stored: InstanceOfName CM_LOOP_DIA
"CM_LOOP_DIA"
BEGIN
END_DATA_BLOCK

DATA_BLOCK "CM_LOOP_HTR_1_DB"   // DB546
{ S7_Optimized_Access := 'FALSE' }
VERSION : 0.0
// stored: InstanceOfName CM_LOOP_HTR_1
"CM_LOOP_HTR_1"
BEGIN
END_DATA_BLOCK

DATA_BLOCK "CM_LOOP_HTR_2_DB"   // DB547
{ S7_Optimized_Access := 'FALSE' }
VERSION : 0.0
// stored: InstanceOfName CM_LOOP_HTR_2
"CM_LOOP_HTR_2"
BEGIN
END_DATA_BLOCK

DATA_BLOCK "CM_LOOP_AVG_SPD_DB"   // DB548
{ S7_Optimized_Access := 'FALSE' }
VERSION : 0.0
// stored: InstanceOfName CM_LOOP_AVG_SPD
"CM_LOOP_AVG_SPD"
BEGIN
END_DATA_BLOCK

DATA_BLOCK "CM_LOOP_MLT_TMP_DB"   // DB549
{ S7_Optimized_Access := 'FALSE' }
VERSION : 0.0
// stored: InstanceOfName CM_LOOP_MLT_TMP
"CM_LOOP_MLT_TMP"
BEGIN
END_DATA_BLOCK

DATA_BLOCK "CM_LOOP_GRW_RTE_DB"   // DB550
{ S7_Optimized_Access := 'FALSE' }
VERSION : 0.0
// stored: InstanceOfName CM_LOOP_GRW_RTE
"CM_LOOP_GRW_RTE"
BEGIN
END_DATA_BLOCK

DATA_BLOCK "CM_LOOP_MLT_LVL_DB"   // DB551
{ S7_Optimized_Access := 'FALSE' }
VERSION : 0.0
// stored: InstanceOfName CM_LOOP_MLT_LVL
"CM_LOOP_MLT_LVL"
BEGIN
END_DATA_BLOCK

DATA_BLOCK "CTL"   // DB552
{ S7_Optimized_Access := 'FALSE' }
VERSION : 0.0
// --------------------------------------------------------------------------------
//     program     :    CTL
//     description :    data for control loops  
//     name        :    G. Eibelsh鋟ser
//     date        :    26.10.2007
// 
//     revision    :
//     name        :
//     date        :    
//                     (c)PVA TePla AG       
//     --------------------------------------------------------------------------------
   VAR
      SET_HTR_1_TMP : Real;   // setpoint for heater 1 temp PID
      SET_HTR_1_MGS_INC : Real;   // heater 1 temperature increment from mgs
      SET_HTR_1_PWR_INC : Real;   // heater 1 power increment from temperature pid controller
      SET_HTR_1_PWR : Real;   // heater 1 power set point
      SET_HTR_2_PWR : Real;   // heater 2 power set point
      SET_XT_SPD : Real;   // xtal speed set point
      SET_CR_SPD : Real;   // crucible speed set point
      SET_CR_ROT : Real;   // crucible rotation set point
      SET_CTL_VALVE_POS : Real;   // control valve position set point
      AVG_MLT_1_TMP : Real;   // average melt 1 temperature
      Y_MLT_1_TMP : Real;   // pid output melt 1 temperature control
      AVG_XT_SPD : Real;   // average xtal speed
      Y_AVG_XT_SPD : Real;   // pid output average speed control
      AVG_CRUC_ROT : Real;   // average crucible rotation
      Y_AVG_CRUC_ROT : Real;   // pid output average crucible rotation control
      ACT_GRW_RTE : Real;   // actual xtal gowth rate
      Y_GRW_RTE : Real;   // pid output growth rate control
      ACT_MLT_LVL : Real;   // actual melt level
      SET_CR_SPD_COF_OFFS : Real;   // actual crucible speed coeffizient offset
      Y_DIA_TMP : Real;   // pid output diamter-temperature controller
      SET_MOB_FDR_VIB_FRQ : Real;
      SET_GAP_CTL_OFFS : Real;   // set point gap offset in [mm], 0 = normal melt lvl
      AVG_GAP_CTL_OFFS : Real;   // average offset gap set point in [mm]
      SET_SPEED_OFFS : Real;   // pid output of offset speed controller for cruc. and xtal lift
      Y_AVG_GAP_OFFS : Real;   // pid output average gap offset in [癈]
   END_VAR
BEGIN
END_DATA_BLOCK

DATA_BLOCK "CRUC"   // DB553
{ S7_Optimized_Access := 'FALSE' }
VERSION : 0.0
// --------------------------------------------------------------------------------
//     program     :    ekz_cm_crucible
//     description :    Calculation of crucible geometry.   
//     name        :    D. Bruess
//     date        :    15.12.99
// 
//     revision    :  
//     name        :
//     date        :
//     
// 
//               (c)CGS         
//     --------------------------------------------------------------------------------
   VAR
      Din : Real;   // inner diameter quarz crucible in mm
      Rt : Real;   // transition radius quarz crucible in mm
      Rb : Real;   // bottom radius quarz crucible in mm
      ym : Real;   // y at transition zylinder in mm
      xm : Real;   // x at transition zylinder in mm
      ys : Real;   // y at transition to bottom in mm
      hmax : Real;   // max fill level in mm
      weight_ym : Real;   // weight till ym
      Vsum : Real;   // volume in mm**3
      ACT_CR_WGT : Real;   // actual weight of remaining charge in crucible
      ACT_BY_WGT_CAL : Real;   // actual calc. weight of this BODY
      ACT_XT_WGT_SUM : Real;   // actual sum of weigth of crystals grown before
      ACT_CR_DIA : Real;   // actual crucible dia. of melt surface
      RATIO : Real;   // calc. value for (v_cr/v_xt)
      BY1_WGT : Real;   // weight of this BODY (saved at end for next one)
      old_qrz_wall_thickness : Real;
      old_qrz_bottom_thickness : Real;
      old_graphite_trans_rad : Real;
      old_graphite_bottom_rad : Real;
      old_graphite_inner_dia : Real;
      old_silicon_charge : Real;
   END_VAR
BEGIN
END_DATA_BLOCK

DATA_BLOCK "CM_LOOP_AVG_CRUC_ROT_DB"   // DB554
{ S7_Optimized_Access := 'FALSE' }
VERSION : 0.0
// stored: InstanceOfName CM_LOOP_AVG_CRUC_ROT
"CM_LOOP_AVG_CRUC_ROT"
BEGIN
END_DATA_BLOCK

DATA_BLOCK "CM_LOOP_GAP_DB"   // DB555
{ S7_Optimized_Access := 'FALSE' }
VERSION : 0.0
// stored: InstanceOfName CM_LOOP_GAP
"CM_LOOP_GAP"
BEGIN
END_DATA_BLOCK

DATA_BLOCK "CM_SEL_CTRL_ALG_DB"   // DB556
{ S7_Optimized_Access := 'FALSE' }
VERSION : 0.0
// stored: InstanceOfName CM_SEL_CTRL_ALG
"CM_SEL_CTRL_ALG"
BEGIN
END_DATA_BLOCK

DATA_BLOCK "CM_CALC_DB"   // DB557
{ S7_Optimized_Access := 'FALSE' }
VERSION : 0.0
// stored: InstanceOfName CM_CALC
"CM_CALC"
BEGIN
END_DATA_BLOCK

DATA_BLOCK "CM_LOOP_AVG_GAP_OFFS_DB"   // DB559
{ S7_Optimized_Access := 'FALSE' }
VERSION : 0.0
// stored: InstanceOfName CM_LOOP_AVG_GAP_OFFS
"CM_LOOP_AVG_GAP_OFFS"
BEGIN
END_DATA_BLOCK

DATA_BLOCK "CM_AVG_MSR_SEN_POS_DB"   // DB560
{ S7_Optimized_Access := 'FALSE' }
VERSION : 0.0
// stored: InstanceOfName CM_AVG_MSR_SEN_POS
"CM_AVG_MSR_SEN_POS"
BEGIN
END_DATA_BLOCK

DATA_BLOCK "CM_LOOP_MLT_DRIFT_DB"   // DB561
{ S7_Optimized_Access := 'FALSE' }
VERSION : 0.0
// stored: InstanceOfName CM_LOOP_MLT_DRIFT
"CM_LOOP_MLT_DRIFT"
BEGIN
END_DATA_BLOCK

DATA_BLOCK "CM_LOOP_DIA_TMP_DB"   // DB562
{ S7_Optimized_Access := 'FALSE' }
VERSION : 0.0
// stored: InstanceOfName CM_LOOP_DIA_TMP
"CM_LOOP_DIA_TMP"
BEGIN
END_DATA_BLOCK

DATA_BLOCK "AM_BY2_RP_CALC_INC_DB"   // DB572
{ S7_Optimized_Access := 'FALSE' }
VERSION : 0.0
// stored: InstanceOfName AM_BY2_RP_CALC_INC
"AM_BY2_RP_CALC_INC"
BEGIN
END_DATA_BLOCK

DATA_BLOCK "AM_PRS_CTRL_DB"   // DB573
{ S7_Optimized_Access := 'FALSE' }
VERSION : 0.0
// stored: InstanceOfName AM_PRS_CTRL
"AM_PRS_CTRL"
BEGIN
END_DATA_BLOCK

DATA_BLOCK "AM_XT_DRV_MOVE_DB"   // DB574
{ S7_Optimized_Access := 'FALSE' }
VERSION : 0.0
// stored: InstanceOfName AM_DRV_MOVE
"AM_DRV_MOVE"
BEGIN
END_DATA_BLOCK

DATA_BLOCK "AM_CR_DRV_MOVE_DB"   // DB575
{ S7_Optimized_Access := 'FALSE' }
VERSION : 0.0
// stored: InstanceOfName AM_DRV_MOVE
"AM_DRV_MOVE"
BEGIN
END_DATA_BLOCK

DATA_BLOCK "AM_CTRL_DB"   // DB576
{ S7_Optimized_Access := 'FALSE' }
VERSION : 0.0
// stored: InstanceOfName AM_CTRL
"AM_CTRL"
BEGIN
END_DATA_BLOCK

DATA_BLOCK "AM_ID_DB"   // DB578
{ S7_Optimized_Access := 'FALSE' }
VERSION : 0.0
// stored: InstanceOfName AM_ID
"AM_ID"
BEGIN
END_DATA_BLOCK

DATA_BLOCK "AM_PD_DB"   // DB579
{ S7_Optimized_Access := 'FALSE' }
VERSION : 0.0
// stored: InstanceOfName AM_PD
"AM_PD"
BEGIN
END_DATA_BLOCK

DATA_BLOCK "AM_ME_DB"   // DB580
{ S7_Optimized_Access := 'FALSE' }
VERSION : 0.0
// stored: InstanceOfName AM_ME
"AM_ME"
BEGIN
END_DATA_BLOCK

DATA_BLOCK "AM_DI_DB"   // DB581
{ S7_Optimized_Access := 'FALSE' }
VERSION : 0.0
// stored: InstanceOfName AM_DI
"AM_DI"
BEGIN
END_DATA_BLOCK

DATA_BLOCK "AM_NE_DB"   // DB582
{ S7_Optimized_Access := 'FALSE' }
VERSION : 0.0
// stored: InstanceOfName AM_NE
"AM_NE"
BEGIN
END_DATA_BLOCK

DATA_BLOCK "AM_SH_DB"   // DB583
{ S7_Optimized_Access := 'FALSE' }
VERSION : 0.0
// stored: InstanceOfName AM_SH
"AM_SH"
BEGIN
END_DATA_BLOCK

DATA_BLOCK "AM_BY_DB"   // DB584
{ S7_Optimized_Access := 'FALSE' }
VERSION : 0.0
// stored: InstanceOfName AM_BY
"AM_BY"
BEGIN
END_DATA_BLOCK

DATA_BLOCK "AM_EC_DB"   // DB585
{ S7_Optimized_Access := 'FALSE' }
VERSION : 0.0
// stored: InstanceOfName AM_EC
"AM_EC"
BEGIN
END_DATA_BLOCK

DATA_BLOCK "AM_SD_DB"   // DB586
{ S7_Optimized_Access := 'FALSE' }
VERSION : 0.0
// stored: InstanceOfName AM_SD
"AM_SD"
BEGIN
END_DATA_BLOCK

DATA_BLOCK "AM_RE_DB"   // DB587
{ S7_Optimized_Access := 'FALSE' }
VERSION : 0.0
// stored: InstanceOfName AM_RE
"AM_RE"
BEGIN
END_DATA_BLOCK

DATA_BLOCK "AM_EMG_DB"   // DB588
{ S7_Optimized_Access := 'FALSE' }
VERSION : 0.0
// stored: InstanceOfName AM_EMG
"AM_EMG"
BEGIN
END_DATA_BLOCK

DATA_BLOCK "BM_MAG_DB"   // DB607
{ S7_Optimized_Access := 'FALSE' }
VERSION : 0.0
// stored: InstanceOfName BM_MAG
"BM_MAG"
BEGIN
END_DATA_BLOCK

DATA_BLOCK "BM_CALL_DRV_DB"   // DB608
{ S7_Optimized_Access := 'FALSE' }
VERSION : 0.0
// stored: InstanceOfName BM_CALL_DRV
"BM_CALL_DRV"
BEGIN
END_DATA_BLOCK

DATA_BLOCK "BM_CALL_HTR_CTRL_DB"   // DB609
{ S7_Optimized_Access := 'FALSE' }
VERSION : 0.0
// stored: InstanceOfName BM_CALL_HTR_CTRL
"BM_CALL_HTR_CTRL"
BEGIN
END_DATA_BLOCK

DATA_BLOCK "BM_CALL_RES_CALC_DB"   // DB612
{ S7_Optimized_Access := 'FALSE' }
VERSION : 0.0
// stored: InstanceOfName BM_CALL_RES_CALC
"BM_CALL_RES_CALC"
BEGIN
END_DATA_BLOCK

DATA_BLOCK "SM_FLT_SETP_DEV_PRC_DB"   // DB613
{ S7_Optimized_Access := 'FALSE' }
VERSION : 0.0
// stored: InstanceOfName SM_FLT_SETP_DEV_PRC
"SM_FLT_SETP_DEV_PRC"
BEGIN
END_DATA_BLOCK

DATA_BLOCK "BM_MCC_DB"   // DB614
{ S7_Optimized_Access := 'FALSE' }
VERSION : 0.0
// stored: InstanceOfName BM_MCC
"BM_MCC"
BEGIN
END_DATA_BLOCK

DATA_BLOCK "BM_XT_WGT_CALC_DB"   // DB615
{ S7_Optimized_Access := 'FALSE' }
VERSION : 0.0
// stored: InstanceOfName BM_XT_WGT_CALC
"BM_XT_WGT_CALC"
BEGIN
END_DATA_BLOCK

DATA_BLOCK "BM_ROT_DRV_DIR_DB"   // DB616
{ S7_Optimized_Access := 'FALSE' }
VERSION : 0.0
// stored: InstanceOfName BM_ROT_DRV_DIR
"BM_ROT_DRV_DIR"
BEGIN
END_DATA_BLOCK

DATA_BLOCK "BM_OP_CALL_DB"   // DB617
{ S7_Optimized_Access := 'FALSE' }
VERSION : 0.0
// stored: InstanceOfName BM_OP_CALL
"BM_OP_CALL"
BEGIN
END_DATA_BLOCK

DATA_BLOCK "BM_S_CAM_EVAL_DB"   // DB618
{ S7_Optimized_Access := 'FALSE' }
VERSION : 0.0
// stored: InstanceOfName BM_S_CAM_EVAL
"BM_S_CAM_EVAL"
BEGIN
END_DATA_BLOCK

DATA_BLOCK "BM_SEED_TMP_CTL_DB"   // DB629
{ S7_Optimized_Access := 'FALSE' }
VERSION : 0.0
// stored: InstanceOfName BM_SEED_TMP_CTL
"BM_SEED_TMP_CTL"
BEGIN
END_DATA_BLOCK

DATA_BLOCK "BM_SI_FIL_REG_DB"   // DB630
{ S7_Optimized_Access := 'FALSE' }
VERSION : 0.0
// stored: InstanceOfName BM_SI_FIL_REG
"BM_SI_FIL_REG"
BEGIN
END_DATA_BLOCK

DATA_BLOCK "BM_XT_HDL_DB"   // DB631
{ S7_Optimized_Access := 'FALSE' }
VERSION : 0.0
// stored: InstanceOfName BM_XT_HDL
"BM_XT_HDL"
BEGIN
END_DATA_BLOCK

DATA_BLOCK "BM_XT_HDL_SEQ_DB"   // DB632
{ S7_Optimized_Access := 'FALSE' }
VERSION : 0.0
// stored: InstanceOfName BM_XT_HDL_SEQ
"BM_XT_HDL_SEQ"
BEGIN
END_DATA_BLOCK

DATA_BLOCK "BM_VSL_HDL_DB"   // DB633
{ S7_Optimized_Access := 'FALSE' }
VERSION : 0.0
// stored: InstanceOfName BM_VSL_HDL
"BM_VSL_HDL"
BEGIN
END_DATA_BLOCK

DATA_BLOCK "BM_VSL_HDL_DRV_DB"   // DB634
{ S7_Optimized_Access := 'FALSE' }
VERSION : 0.0
// stored: InstanceOfName BM_VSL_HDL_DRV
"BM_VSL_HDL_DRV"
BEGIN
END_DATA_BLOCK

DATA_BLOCK "BM_CDP_DB"   // DB636
{ S7_Optimized_Access := 'FALSE' }
VERSION : 0.0
// stored: InstanceOfName BM_CDP
"BM_CDP"
BEGIN
END_DATA_BLOCK

DATA_BLOCK "BM_MLT_VIB_MON_DB"   // DB637
{ S7_Optimized_Access := 'FALSE' }
VERSION : 0.0
// stored: InstanceOfName BM_MLT_VIB_MON
"BM_MLT_VIB_MON"
BEGIN
END_DATA_BLOCK

DATA_BLOCK "BM_XT_ORB_DET_DB"   // DB638
{ S7_Optimized_Access := 'FALSE' }
VERSION : 0.0
// stored: InstanceOfName BM_XT_ORB_DET
"BM_XT_ORB_DET"
BEGIN
END_DATA_BLOCK

DATA_BLOCK "BM_MLT_LVL_MON_DB"   // DB639
{ S7_Optimized_Access := 'FALSE' }
VERSION : 0.0
// stored: InstanceOfName BM_MLT_LVL_MON
"BM_MLT_LVL_MON"
BEGIN
END_DATA_BLOCK

DATA_BLOCK "BM_CALL_CAM_DB"   // DB640
{ S7_Optimized_Access := 'FALSE' }
VERSION : 0.0
// stored: InstanceOfName BM_CALL_CAM
"BM_CALL_CAM"
BEGIN
END_DATA_BLOCK

DATA_BLOCK "BM_CAM_RECV_DB"   // DB641
{ S7_Optimized_Access := 'FALSE' }
VERSION : 0.0
// --------------------------------------------------------------------------------
//     program     :    BM_CAM_RECV_DB
//     description :    camera receive data      
//     name        :    G. Eibelsh鋟ser
//     date        :    03.05.2010
// 
//     revision    :
//     name        :
//     date        :    
//                     (c)PVA Tepla AG
//     --------------------------------------------------------------------------------
   VAR
      Data : Array[0..255] of Char;
   END_VAR
BEGIN
END_DATA_BLOCK

DATA_BLOCK "BM_CAM_EVAL_DB"   // DB642
{ S7_Optimized_Access := 'FALSE' }
VERSION : 0.0
// --------------------------------------------------------------------------------
//     program     :    BM_CAM_EVAL_DB
//     description :    camera evaluation data     
//     name        :    G. Eibelsh鋟ser
//     date        :    03.05.2010
// 
//     revision    :
//     name        :
//     date        :    
//                     (c)PVA Tepla AG
//     --------------------------------------------------------------------------------
   VAR
      Data : Array[0..255] of Char;
   END_VAR
BEGIN
END_DATA_BLOCK

DATA_BLOCK "BM_MOB_FDR_MAIN_DB"   // DB643
{ S7_Optimized_Access := 'FALSE' }
VERSION : 0.0
// stored: InstanceOfName BM_MOB_FDR_MAIN
"BM_MOB_FDR_MAIN"
BEGIN
END_DATA_BLOCK

DATA_BLOCK "BM_MOB_FDR_DCK_DB"   // DB644
{ S7_Optimized_Access := 'FALSE' }
VERSION : 0.0
// stored: InstanceOfName BM_MOB_FDR_DCK
"BM_MOB_FDR_DCK"
BEGIN
END_DATA_BLOCK

DATA_BLOCK "BM_MOB_FDR_UDCK_DB"   // DB645
{ S7_Optimized_Access := 'FALSE' }
VERSION : 0.0
// stored: InstanceOfName BM_MOB_FDR_UDCK
"BM_MOB_FDR_UDCK"
BEGIN
END_DATA_BLOCK

DATA_BLOCK "BM_MOB_FDR_DRV_SEQ_DB"   // DB646
{ S7_Optimized_Access := 'FALSE' }
VERSION : 0.0
// stored: InstanceOfName BM_MOB_FDR_DRV_SEQ
"BM_MOB_FDR_DRV_SEQ"
BEGIN
END_DATA_BLOCK

DATA_BLOCK "BM_ACC_MAIN_DB"   // DB649
{ S7_Optimized_Access := 'FALSE' }
VERSION : 0.0
// stored: InstanceOfName BM_ACC_MAIN
"BM_ACC_MAIN"
BEGIN
END_DATA_BLOCK

DATA_BLOCK "BM_ACC_PRS_MON_DB"   // DB650
{ S7_Optimized_Access := 'FALSE' }
VERSION : 0.0
// stored: InstanceOfName BM_ACC_PRS_MON
"BM_ACC_PRS_MON"
BEGIN
END_DATA_BLOCK

